C07281=1014.673,-56.612,386.212,-24.068,21.603,-43.637
C07282=1014.673,-56.279,386.186,-24.068,21.603,-43.632
C07283=1014.675,-55.946,386.161,-24.069,21.603,-43.627
C07284=1014.675,-55.613,386.136,-24.070,21.602,-43.623
C07285=1014.676,-55.280,386.111,-24.070,21.602,-43.618
C07286=1014.676,-54.948,386.085,-24.071,21.601,-43.613
C07287=1014.677,-54.616,386.060,-24.072,21.601,-43.608
C07288=1014.678,-54.284,386.034,-24.072,21.600,-43.603
C07289=1014.679,-53.951,386.010,-24.073,21.599,-43.599
C07290=1014.679,-53.619,385.984,-24.074,21.600,-43.594
C07291=1014.680,-53.287,385.959,-24.074,21.598,-43.589
C07292=1014.680,-52.954,385.933,-24.075,21.598,-43.584
C07293=1014.681,-52.622,385.909,-24.075,21.597,-43.579
C07294=1014.681,-52.290,385.883,-24.076,21.597,-43.575
C07295=1014.682,-51.957,385.857,-24.077,21.597,-43.570
C07296=1014.683,-51.625,385.832,-24.077,21.596,-43.566
C07297=1014.683,-51.293,385.806,-24.078,21.596,-43.560
C07298=1014.683,-50.960,385.781,-24.079,21.595,-43.555
C07299=1014.684,-50.628,385.756,-24.079,21.594,-43.551
C07300=1014.684,-50.296,385.731,-24.080,21.595,-43.546
C07301=1014.685,-49.963,385.705,-24.080,21.593,-43.542
C07302=1014.685,-49.630,385.680,-24.081,21.593,-43.536
C07303=1014.686,-49.298,385.654,-24.081,21.592,-43.532
C07304=1014.686,-48.966,385.629,-24.082,21.592,-43.527
C07305=1014.686,-48.633,385.604,-24.083,21.592,-43.522
C07306=1014.686,-48.301,385.578,-24.083,21.591,-43.518
C07307=1014.687,-47.968,385.552,-24.084,21.591,-43.512
C07308=1014.687,-47.635,385.527,-24.085,21.589,-43.508
C07309=1014.687,-47.303,385.501,-24.086,21.589,-43.503
C07310=1014.688,-46.971,385.476,-24.086,21.590,-43.498
C07311=1014.688,-46.639,385.450,-24.087,21.588,-43.494
C07312=1014.688,-46.306,385.425,-24.088,21.588,-43.488
C07313=1014.689,-45.973,385.399,-24.088,21.588,-43.485
C07314=1014.689,-45.641,385.373,-24.089,21.587,-43.479
C07315=1014.689,-45.308,385.348,-24.089,21.586,-43.475
C07316=1014.689,-44.976,385.323,-24.090,21.586,-43.470
C07317=1014.688,-44.643,385.296,-24.091,21.586,-43.465
C07318=1014.688,-44.310,385.271,-24.091,21.585,-43.461
C07319=1014.689,-43.978,385.246,-24.092,21.585,-43.455
C07320=1014.689,-43.645,385.220,-24.092,21.584,-43.451
C07321=1014.689,-43.312,385.195,-24.093,21.583,-43.446
C07322=1014.689,-42.980,385.168,-24.094,21.583,-43.442
C07323=1014.689,-42.648,385.143,-24.094,21.583,-43.437
C07324=1014.689,-42.315,385.118,-24.095,21.582,-43.431
C07325=1014.688,-41.982,385.091,-24.096,21.582,-43.427
C07326=1014.689,-41.650,385.066,-24.096,21.582,-43.422
C07327=1014.689,-41.317,385.041,-24.097,21.580,-43.418
C07328=1014.688,-40.985,385.015,-24.098,21.580,-43.413
C07329=1014.689,-40.652,384.988,-24.098,21.580,-43.409
C07330=1014.688,-40.319,384.963,-24.099,21.579,-43.404
C07331=1014.688,-39.987,384.937,-24.100,21.579,-43.398
C07332=1014.688,-39.654,384.911,-24.100,21.578,-43.394
C07333=1014.688,-39.321,384.886,-24.101,21.578,-43.389
C07334=1014.687,-38.989,384.860,-24.101,21.577,-43.385
C07335=1014.687,-38.657,384.834,-24.102,21.577,-43.380
C07336=1014.687,-38.323,384.808,-24.102,21.576,-43.376
C07337=1014.687,-37.991,384.783,-24.103,21.576,-43.371
C07338=1014.686,-37.658,384.757,-24.104,21.575,-43.366
C07339=1014.686,-37.326,384.731,-24.105,21.575,-43.361
C07340=1014.686,-36.993,384.705,-24.105,21.574,-43.357
C07341=1014.685,-36.660,384.680,-24.106,21.574,-43.352
C07342=1014.684,-36.328,384.653,-24.107,21.574,-43.347
C07343=1014.685,-35.995,384.628,-24.107,21.573,-43.343
C07344=1014.684,-35.662,384.602,-24.108,21.573,-43.337
C07345=1014.683,-35.330,384.576,-24.108,21.572,-43.334
C07346=1014.683,-34.997,384.549,-24.109,21.572,-43.328
C07347=1014.683,-34.664,384.525,-24.109,21.571,-43.324
C07348=1014.682,-34.332,384.498,-24.110,21.571,-43.319
C07349=1014.682,-33.999,384.472,-24.111,21.570,-43.315
C07350=1014.681,-33.666,384.446,-24.111,21.570,-43.310
C07351=1014.680,-33.334,384.420,-24.112,21.569,-43.306
C07352=1014.680,-33.001,384.395,-24.113,21.569,-43.301
C07353=1014.679,-32.668,384.368,-24.113,21.568,-43.296
C07354=1014.679,-32.336,384.342,-24.114,21.568,-43.291
C07355=1014.678,-32.002,384.316,-24.114,21.567,-43.287
C07356=1014.677,-31.670,384.290,-24.115,21.567,-43.282
C07357=1014.677,-31.337,384.264,-24.116,21.566,-43.278
C07358=1014.676,-31.004,384.238,-24.116,21.566,-43.273
C07359=1014.675,-30.672,384.212,-24.117,21.565,-43.269
C07360=1014.675,-30.339,384.186,-24.118,21.565,-43.264
C07361=1014.674,-30.006,384.160,-24.118,21.565,-43.260
C07362=1014.674,-29.674,384.134,-24.119,21.564,-43.254
C07363=1014.673,-29.340,384.108,-24.119,21.563,-43.250
C07364=1014.672,-29.008,384.081,-24.120,21.563,-43.245
C07365=1014.671,-28.675,384.055,-24.120,21.562,-43.241
C07366=1014.670,-28.342,384.030,-24.121,21.562,-43.236
C07367=1014.669,-28.010,384.004,-24.122,21.562,-43.232
C07368=1014.669,-27.678,383.977,-24.123,21.562,-43.227
C07369=1014.667,-27.344,383.951,-24.123,21.560,-43.223
C07370=1014.667,-27.012,383.925,-24.124,21.560,-43.217
C07371=1014.666,-26.679,383.899,-24.124,21.560,-43.214
C07372=1014.664,-26.346,383.872,-24.125,21.559,-43.208
C07373=1014.664,-26.013,383.846,-24.126,21.559,-43.204
C07374=1014.663,-25.680,383.821,-24.126,21.559,-43.199
C07375=1014.661,-25.348,383.794,-24.127,21.558,-43.195
C07376=1014.661,-25.015,383.768,-24.128,21.558,-43.190
C07377=1014.659,-24.682,383.742,-24.128,21.557,-43.186
C07378=1014.659,-24.349,383.715,-24.129,21.557,-43.181
C07379=1014.657,-24.017,383.688,-24.129,21.556,-43.177
C07380=1014.657,-23.683,383.663,-24.130,21.556,-43.171
C07381=1014.655,-23.351,383.636,-24.131,21.555,-43.168
C07382=1014.654,-23.018,383.611,-24.131,21.556,-43.162
C07383=1014.653,-22.685,383.584,-24.132,21.554,-43.158
C07384=1014.652,-22.353,383.558,-24.133,21.554,-43.153
C07385=1014.651,-22.019,383.531,-24.133,21.554,-43.149
C07386=1014.649,-21.687,383.505,-24.134,21.553,-43.144
C07387=1014.648,-21.355,383.479,-24.134,21.552,-43.140
C07388=1014.647,-21.021,383.453,-24.135,21.553,-43.135
C07389=1014.645,-20.689,383.426,-24.136,21.552,-43.131
C07390=1014.644,-20.356,383.400,-24.136,21.551,-43.127
C07391=1014.643,-20.023,383.374,-24.137,21.551,-43.122
C07392=1014.642,-19.851,383.360,-24.137,21.550,-43.118
C07393=1014.640,-19.434,383.327,-24.138,21.550,-43.112
C07394=1014.640,-19.187,383.307,-24.139,21.550,-43.109
C07395=1014.638,-18.925,383.286,-24.139,21.550,-43.107
C07396=1014.637,-18.663,383.266,-24.139,21.549,-43.105
C07397=1014.637,-18.416,383.246,-24.139,21.548,-43.103
C07398=1014.635,-18.194,383.228,-24.140,21.549,-43.100
C07399=1014.634,-17.829,383.200,-24.141,21.548,-43.092
C07400=1014.632,-17.496,383.173,-24.141,21.547,-43.088
C07401=1014.631,-17.163,383.146,-24.142,21.547,-43.083
C07402=1014.630,-16.830,383.120,-24.142,21.547,-43.079
C07403=1014.628,-16.497,383.093,-24.143,21.546,-43.074
C07404=1014.626,-16.162,383.067,-24.144,21.546,-43.070
C07405=1014.624,-15.827,383.040,-24.145,21.546,-43.065
C07406=1014.623,-15.491,383.014,-24.145,21.545,-43.061
C07407=1014.621,-15.152,382.986,-24.146,21.544,-43.055
C07408=1014.619,-14.812,382.960,-24.146,21.544,-43.052
C07409=1014.618,-14.471,382.932,-24.147,21.544,-43.046
C07410=1014.616,-14.127,382.905,-24.147,21.543,-43.042
C07411=1014.615,-13.780,382.877,-24.148,21.543,-43.037
C07412=1014.613,-13.432,382.849,-24.149,21.542,-43.033
C07413=1014.611,-13.081,382.822,-24.149,21.542,-43.028
C07414=1014.609,-12.729,382.793,-24.150,21.541,-43.024
C07415=1014.607,-12.376,382.765,-24.151,21.541,-43.019
C07416=1014.606,-12.021,382.737,-24.151,21.540,-43.014
C07417=1014.604,-11.664,382.708,-24.152,21.540,-43.009
C07418=1014.602,-11.306,382.680,-24.152,21.539,-43.006
C07419=1014.599,-10.948,382.651,-24.153,21.539,-43.000
C07420=1014.598,-10.588,382.623,-24.154,21.539,-42.995
C07421=1014.596,-10.227,382.593,-24.154,21.538,-42.991
C07422=1014.594,-9.866,382.564,-24.155,21.538,-42.985
C07423=1014.592,-9.504,382.535,-24.156,21.537,-42.982
C07424=1014.589,-9.142,382.506,-24.156,21.536,-42.976
C07425=1014.587,-8.778,382.477,-24.157,21.536,-42.971
C07426=1014.585,-8.416,382.448,-24.158,21.536,-42.967
C07427=1014.583,-8.053,382.419,-24.158,21.535,-42.961
C07428=1014.580,-7.686,382.390,-24.159,21.535,-42.956
C07429=1014.578,-7.317,382.361,-24.160,21.534,-42.952
C07430=1014.576,-6.945,382.330,-24.160,21.534,-42.947
C07431=1014.574,-6.571,382.300,-24.161,21.533,-42.941
C07432=1014.572,-6.196,382.270,-24.162,21.533,-42.937
C07433=1014.568,-5.820,382.240,-24.163,21.533,-42.932
C07434=1014.567,-5.447,382.210,-24.163,21.532,-42.928
C07435=1014.564,-5.076,382.180,-24.164,21.532,-42.923
C07436=1014.561,-4.710,382.150,-24.164,21.531,-42.919
C07437=1014.559,-4.349,382.122,-24.165,21.530,-42.913
C07438=1014.556,-3.991,382.092,-24.166,21.531,-42.908
C07439=1014.554,-3.637,382.065,-24.166,21.529,-42.904
C07440=1014.552,-3.285,382.036,-24.167,21.529,-42.899
C07441=1014.549,-2.933,382.007,-24.167,21.529,-42.895
C07442=1014.547,-2.583,381.979,-24.168,21.529,-42.890
C07443=1014.545,-2.236,381.951,-24.169,21.528,-42.886
C07444=1014.542,-1.888,381.923,-24.169,21.528,-42.880
C07445=1014.540,-1.544,381.896,-24.170,21.527,-42.877
C07446=1014.537,-1.201,381.868,-24.170,21.527,-42.873
C07447=1014.535,-0.858,381.840,-24.171,21.526,-42.867
C07448=1014.532,-0.519,381.813,-24.172,21.526,-42.864
C07449=1014.529,-0.180,381.785,-24.172,21.526,-42.858
C07450=1014.527,0.157,381.759,-24.173,21.525,-42.855
C07451=1014.525,0.493,381.731,-24.173,21.525,-42.851
C07452=1014.522,0.827,381.704,-24.174,21.525,-42.846
C07453=1014.519,1.161,381.677,-24.175,21.524,-42.842
C07454=1014.516,1.495,381.650,-24.175,21.523,-42.838
C07455=1014.514,1.825,381.623,-24.176,21.523,-42.834
C07456=1014.512,2.138,381.598,-24.176,21.523,-42.831
C07457=1014.509,2.426,381.574,-24.177,21.522,-42.827
C07458=1014.508,2.695,381.553,-24.177,21.522,-42.823
C07459=1014.505,2.957,381.532,-24.178,21.522,-42.818
C07460=1014.503,3.226,381.510,-24.179,21.521,-42.814
C07461=1014.500,3.515,381.487,-24.179,21.521,-42.810
C07462=1014.498,3.829,381.461,-24.179,21.520,-42.807
C07463=1014.496,4.158,381.434,-24.180,21.521,-42.803
C07464=1014.493,4.490,381.408,-24.180,21.519,-42.799
C07465=1014.490,4.821,381.380,-24.181,21.519,-42.795
C07466=1014.487,5.151,381.354,-24.181,21.518,-42.792
C07467=1014.485,5.481,381.327,-24.182,21.519,-42.786
C07468=1014.481,5.811,381.300,-24.183,21.518,-42.783
C07469=1014.479,6.141,381.273,-24.183,21.518,-42.779
C07470=1014.475,6.470,381.247,-24.184,21.518,-42.774
C07471=1014.473,6.798,381.220,-24.185,21.517,-42.770
C07472=1014.470,7.126,381.193,-24.185,21.517,-42.766
C07473=1014.467,7.451,381.167,-24.186,21.516,-42.762
C07474=1014.464,7.775,381.141,-24.186,21.516,-42.759
C07475=1014.462,8.095,381.114,-24.186,21.515,-42.755
C07476=1014.459,8.413,381.088,-24.187,21.516,-42.750
C07477=1014.456,8.729,381.063,-24.188,21.515,-42.746
C07478=1014.453,9.044,381.037,-24.188,21.515,-42.742
C07479=1014.450,9.359,381.011,-24.189,21.514,-42.738
C07480=1014.448,9.673,380.986,-24.190,21.514,-42.733
C07481=1014.444,9.989,380.961,-24.190,21.514,-42.730
C07482=1014.442,10.306,380.934,-24.191,21.513,-42.726
C07483=1014.438,10.625,380.909,-24.191,21.513,-42.722
C07484=1014.435,10.945,380.883,-24.192,21.512,-42.718
C07485=1014.432,11.267,380.856,-24.192,21.512,-42.715
C07486=1014.429,11.591,380.830,-24.193,21.511,-42.711
C07487=1014.426,11.914,380.803,-24.193,21.511,-42.707
C07488=1014.423,12.237,380.777,-24.194,21.511,-42.702
C07489=1014.420,12.561,380.751,-24.194,21.510,-42.698
C07490=1014.416,12.885,380.724,-24.195,21.510,-42.694
C07491=1014.413,13.208,380.698,-24.195,21.509,-42.691
C07492=1014.410,13.533,380.671,-24.196,21.509,-42.687
C07493=1014.406,13.857,380.645,-24.197,21.509,-42.682
C07494=1014.403,14.181,380.618,-24.197,21.509,-42.678
C07495=1014.400,14.506,380.591,-24.198,21.508,-42.674
C07496=1014.396,14.832,380.566,-24.198,21.508,-42.670
C07497=1014.393,15.158,380.539,-24.199,21.507,-42.667
C07498=1014.390,15.484,380.512,-24.199,21.507,-42.663
C07499=1014.387,15.811,380.485,-24.200,21.507,-42.658
C07500=1014.383,16.139,380.458,-24.200,21.506,-42.654
C07501=1014.380,16.467,380.431,-24.201,21.506,-42.650
C07502=1014.376,16.795,380.405,-24.201,21.505,-42.646
C07503=1014.372,17.124,380.378,-24.202,21.505,-42.643
C07504=1014.370,17.454,380.351,-24.202,21.504,-42.639
C07505=1014.366,17.784,380.324,-24.203,21.504,-42.634
C07506=1014.362,18.115,380.296,-24.204,21.504,-42.630
C07507=1014.358,18.446,380.270,-24.204,21.503,-42.626
C07508=1014.354,18.778,380.243,-24.205,21.503,-42.622
C07509=1014.352,19.110,380.215,-24.205,21.502,-42.619
C07510=1014.347,19.458,380.187,-24.206,21.503,-42.613
C07511=1014.342,19.875,380.152,-24.207,21.502,-42.608
C07512=1014.340,20.112,380.133,-24.207,21.502,-42.604
C07513=1014.338,20.358,380.113,-24.207,21.502,-42.603
C07514=1014.334,20.606,380.093,-24.208,21.502,-42.601
C07515=1014.332,20.848,380.073,-24.208,21.502,-42.599
C07516=1014.329,21.075,380.054,-24.208,21.501,-42.597
C07517=1014.327,21.282,380.037,-24.209,21.501,-42.593
C07518=1014.322,21.639,380.008,-24.209,21.500,-42.588
C07519=1014.319,21.962,379.981,-24.210,21.501,-42.584
C07520=1014.315,22.256,379.957,-24.210,21.500,-42.582
C07521=1014.312,22.509,379.936,-24.210,21.499,-42.580
C07522=1014.307,22.919,379.903,-24.211,21.499,-42.573
C07523=1014.303,23.327,379.869,-24.212,21.498,-42.565
C07524=1014.300,23.579,379.849,-24.213,21.498,-42.562
C07525=1014.296,23.873,379.825,-24.213,21.498,-42.560
C07526=1014.292,24.200,379.798,-24.213,21.497,-42.558
C07527=1014.288,24.534,379.770,-24.214,21.497,-42.553
C07528=1014.284,24.868,379.742,-24.215,21.497,-42.549
C07529=1014.280,25.202,379.715,-24.215,21.496,-42.545
C07530=1014.276,25.537,379.688,-24.216,21.496,-42.541
C07531=1014.271,25.870,379.660,-24.216,21.495,-42.538
C07532=1014.268,26.205,379.632,-24.217,21.495,-42.534
C07533=1014.263,26.539,379.605,-24.217,21.494,-42.530
C07534=1014.259,26.873,379.577,-24.218,21.494,-42.525
C07535=1014.254,27.208,379.550,-24.219,21.495,-42.522
C07536=1014.251,27.542,379.522,-24.219,21.494,-42.518
C07537=1014.246,27.876,379.495,-24.220,21.494,-42.514
C07538=1014.242,28.211,379.468,-24.220,21.493,-42.510
C07539=1014.238,28.545,379.440,-24.221,21.493,-42.507
C07540=1014.233,28.879,379.413,-24.221,21.492,-42.503
C07541=1014.229,29.214,379.385,-24.222,21.493,-42.498
C07542=1014.224,29.548,379.358,-24.222,21.492,-42.494
C07543=1014.220,29.882,379.330,-24.223,21.492,-42.490
C07544=1014.216,30.216,379.302,-24.223,21.491,-42.486
C07545=1014.211,30.551,379.274,-24.224,21.491,-42.483
C07546=1014.207,30.885,379.247,-24.224,21.490,-42.479
C07547=1014.203,31.220,379.220,-24.225,21.490,-42.475
C07548=1014.197,31.555,379.192,-24.225,21.489,-42.471
C07549=1014.193,31.888,379.165,-24.226,21.489,-42.468
C07550=1014.189,32.224,379.137,-24.226,21.489,-42.464
C07551=1014.184,32.558,379.109,-24.227,21.489,-42.459
C07552=1014.180,32.893,379.082,-24.228,21.489,-42.455
C07553=1014.174,33.227,379.054,-24.228,21.488,-42.452
C07554=1014.170,33.561,379.027,-24.229,21.488,-42.448
C07555=1014.165,33.896,378.999,-24.229,21.487,-42.444
C07556=1014.161,34.230,378.971,-24.230,21.487,-42.440
C07557=1014.155,34.565,378.944,-24.230,21.486,-42.437
C07558=1014.151,34.899,378.915,-24.231,21.486,-42.433
C07559=1014.146,35.234,378.889,-24.231,21.485,-42.429
C07560=1014.141,35.569,378.861,-24.232,21.486,-42.426
C07561=1014.136,35.903,378.834,-24.232,21.485,-42.422
C07562=1014.131,36.237,378.806,-24.233,21.485,-42.418
C07563=1014.126,36.573,378.778,-24.234,21.485,-42.413
C07564=1014.121,36.907,378.750,-24.234,21.485,-42.409
C07565=1014.117,37.241,378.723,-24.235,21.484,-42.405
C07566=1014.112,37.576,378.695,-24.235,21.484,-42.402
C07567=1014.106,37.911,378.668,-24.236,21.483,-42.398
C07568=1014.101,38.246,378.640,-24.236,21.483,-42.395
C07569=1014.096,38.580,378.612,-24.237,21.483,-42.391
C07570=1014.092,38.915,378.585,-24.237,21.483,-42.387
C07571=1014.086,39.249,378.557,-24.238,21.482,-42.383
C07572=1014.081,39.584,378.530,-24.238,21.482,-42.380
C07573=1014.076,39.919,378.502,-24.239,21.481,-42.376
C07574=1014.071,40.253,378.474,-24.239,21.481,-42.372
C07575=1014.066,40.588,378.446,-24.240,21.481,-42.369
C07576=1014.060,40.923,378.419,-24.240,21.481,-42.365
C07577=1014.055,41.257,378.391,-24.241,21.480,-42.361
C07578=1014.049,41.592,378.364,-24.241,21.480,-42.357
C07579=1014.045,41.927,378.336,-24.242,21.479,-42.354
C07580=1014.038,42.262,378.308,-24.242,21.479,-42.350
C07581=1014.033,42.596,378.280,-24.243,21.479,-42.347
C07582=1014.028,42.931,378.252,-24.243,21.479,-42.343
C07583=1014.022,43.265,378.225,-24.244,21.478,-42.339
C07584=1014.017,43.600,378.198,-24.244,21.478,-42.335
C07585=1014.012,43.935,378.170,-24.245,21.477,-42.332
C07586=1014.006,44.270,378.142,-24.245,21.477,-42.328
C07587=1014.001,44.605,378.114,-24.246,21.477,-42.325
C07588=1013.995,44.940,378.087,-24.246,21.477,-42.321
C07589=1013.989,45.275,378.059,-24.247,21.476,-42.317
C07590=1013.984,45.609,378.031,-24.247,21.476,-42.313
C07591=1013.978,45.944,378.004,-24.248,21.475,-42.309
C07592=1013.972,46.279,377.976,-24.248,21.475,-42.306
C07593=1013.967,46.613,377.948,-24.249,21.475,-42.302
C07594=1013.961,46.948,377.921,-24.249,21.475,-42.299
C07595=1013.955,47.283,377.893,-24.250,21.474,-42.295
C07596=1013.950,47.618,377.865,-24.250,21.474,-42.291
C07597=1013.943,47.953,377.837,-24.251,21.473,-42.287
C07598=1013.938,48.287,377.810,-24.251,21.473,-42.284
C07599=1013.932,48.623,377.782,-24.252,21.473,-42.280
C07600=1013.926,48.957,377.755,-24.252,21.473,-42.277
C07601=1013.920,49.292,377.727,-24.253,21.472,-42.273
C07602=1013.913,49.627,377.699,-24.253,21.472,-42.269
C07603=1013.908,49.961,377.672,-24.254,21.472,-42.266
C07604=1013.902,50.296,377.644,-24.254,21.471,-42.262
C07605=1013.896,50.631,377.616,-24.255,21.471,-42.258
C07606=1013.890,50.966,377.589,-24.255,21.471,-42.254
C07607=1013.884,51.301,377.561,-24.256,21.471,-42.251
C07608=1013.877,51.636,377.533,-24.256,21.470,-42.247
C07609=1013.871,51.970,377.506,-24.257,21.470,-42.244
C07610=1013.865,52.305,377.478,-24.257,21.470,-42.240
C07611=1013.859,52.641,377.450,-24.258,21.469,-42.238
C07612=1013.852,52.975,377.423,-24.258,21.469,-42.234
C07613=1013.846,53.310,377.395,-24.259,21.468,-42.230
C07614=1013.840,53.645,377.367,-24.259,21.468,-42.227
C07615=1013.816,54.896,377.264,-24.271,21.503,-42.191
C07616=1013.815,54.977,377.257,-24.281,21.541,-42.167
C07617=1013.807,55.373,377.225,-24.331,21.722,-42.052
C07618=1013.799,55.768,377.192,-24.380,21.904,-41.938
C07619=1013.792,56.164,377.159,-24.428,22.086,-41.824
C07620=1013.784,56.560,377.127,-24.477,22.269,-41.710
C07621=1013.776,56.955,377.094,-24.525,22.453,-41.598
C07622=1013.769,57.351,377.061,-24.572,22.637,-41.485
C07623=1013.760,57.747,377.029,-24.620,22.823,-41.372
C07624=1013.753,58.143,376.996,-24.667,23.008,-41.261
C07625=1013.745,58.538,376.963,-24.715,23.195,-41.149
C07626=1013.737,58.934,376.931,-24.761,23.381,-41.038
C07627=1013.730,59.330,376.898,-24.808,23.569,-40.927
C07628=1013.722,59.726,376.866,-24.853,23.757,-40.818
C07629=1013.714,60.121,376.833,-24.899,23.946,-40.708
C07630=1013.706,60.518,376.801,-24.945,24.135,-40.598
C07631=1013.699,60.913,376.768,-24.990,24.326,-40.489
C07632=1013.690,61.309,376.736,-25.035,24.517,-40.381
C07633=1013.683,61.704,376.704,-25.080,24.707,-40.272
C07634=1013.675,62.102,376.671,-25.124,24.901,-40.164
C07635=1013.669,62.386,376.647,-25.156,25.038,-40.089
C07636=1013.665,62.605,376.629,-25.180,25.145,-40.028
C07637=1013.659,62.847,376.610,-25.207,25.264,-39.964
C07638=1013.654,63.095,376.589,-25.234,25.384,-39.898
C07639=1013.650,63.330,376.570,-25.260,25.499,-39.835
C07640=1013.646,63.542,376.553,-25.283,25.603,-39.779
C07641=1013.643,63.947,376.517,-25.297,25.665,-39.741
C07642=1013.642,64.165,376.495,-25.299,25.671,-39.736
C07643=1013.641,64.392,376.475,-25.300,25.677,-39.731
C07644=1013.641,64.619,376.454,-25.302,25.682,-39.725
C07645=1013.640,64.840,376.432,-25.303,25.688,-39.721
C07646=1013.639,65.060,376.413,-25.304,25.693,-39.715
C07647=1013.638,65.275,376.392,-25.306,25.699,-39.711
C07648=1013.638,65.483,376.373,-25.307,25.703,-39.706
C07649=1013.637,65.875,376.335,-25.310,25.713,-39.697
C07650=1013.635,66.203,376.304,-25.312,25.721,-39.689
C07651=1013.634,66.566,376.270,-25.314,25.731,-39.681
C07652=1013.633,66.963,376.233,-25.317,25.740,-39.672
C07653=1013.631,67.362,376.196,-25.319,25.750,-39.663
C07654=1013.630,67.763,376.158,-25.322,25.760,-39.654
C07655=1013.628,68.173,376.120,-25.325,25.771,-39.645
C07656=1013.626,68.591,376.080,-25.328,25.781,-39.635
C07657=1013.626,69.007,376.041,-25.330,25.792,-39.626
C07658=1013.624,69.416,376.002,-25.333,25.803,-39.615
C07659=1013.622,69.819,375.964,-25.336,25.813,-39.606
C07660=1013.621,70.224,375.926,-25.338,25.823,-39.597
C07661=1013.620,70.628,375.888,-25.341,25.832,-39.588
C07662=1013.618,71.032,375.849,-25.343,25.843,-39.579
C07663=1013.617,71.437,375.812,-25.346,25.854,-39.569
C07664=1013.616,71.842,375.773,-25.349,25.865,-39.560
C07665=1013.614,72.248,375.735,-25.352,25.876,-39.550
C07666=1013.612,72.656,375.696,-25.354,25.886,-39.541
C07667=1013.611,73.065,375.657,-25.357,25.896,-39.532
C07668=1013.609,73.476,375.618,-25.360,25.907,-39.522
C07669=1013.608,73.891,375.579,-25.363,25.919,-39.512
C07670=1013.608,74.110,375.558,-25.364,25.923,-39.507
C07671=1013.606,74.338,375.536,-25.366,25.931,-39.502
C07672=1013.606,74.565,375.514,-25.367,25.936,-39.498
C07673=1013.605,74.780,375.495,-25.369,25.941,-39.492
C07674=1013.605,74.989,375.475,-25.370,25.947,-39.488
C07675=1013.603,75.403,375.435,-25.373,25.958,-39.477
C07676=1013.601,75.812,375.397,-25.376,25.970,-39.467
C07677=1013.600,76.214,375.358,-25.378,25.980,-39.458
C07678=1013.599,76.607,375.321,-25.381,25.990,-39.450
C07679=1013.597,76.994,375.284,-25.384,26.001,-39.441
C07680=1013.595,77.376,375.247,-25.386,26.011,-39.432
C07681=1013.594,77.757,375.211,-25.389,26.022,-39.423
C07682=1013.593,78.141,375.175,-25.392,26.033,-39.413
C07683=1013.591,78.530,375.138,-25.394,26.043,-39.404
C07684=1013.590,78.925,375.100,-25.397,26.053,-39.395
C07685=1013.588,79.326,375.061,-25.400,26.065,-39.385
C07686=1013.586,79.735,375.023,-25.402,26.076,-39.377
C07687=1013.585,80.147,374.983,-25.405,26.087,-39.367
C07688=1013.584,80.530,374.947,-25.408,26.098,-39.358
C07689=1013.582,80.893,374.912,-25.410,26.108,-39.349
C07690=1013.580,81.287,374.874,-25.413,26.119,-39.340
C07691=1013.579,81.701,374.835,-25.416,26.131,-39.330
C07692=1013.577,82.115,374.795,-25.419,26.143,-39.321
C07693=1013.576,82.528,374.755,-25.422,26.154,-39.311
C07694=1013.574,82.940,374.717,-25.425,26.165,-39.300
C07695=1013.572,83.351,374.677,-25.428,26.177,-39.291
C07696=1013.571,83.760,374.637,-25.431,26.189,-39.281
C07697=1013.569,84.168,374.599,-25.433,26.200,-39.272
C07698=1013.567,84.575,374.559,-25.436,26.212,-39.263
C07699=1013.566,84.981,374.521,-25.439,26.224,-39.253
C07700=1013.565,85.385,374.482,-25.442,26.236,-39.243
C07701=1013.563,85.788,374.442,-25.445,26.248,-39.233
C07702=1013.561,86.189,374.404,-25.447,26.259,-39.225
C07703=1013.560,86.591,374.366,-25.450,26.271,-39.215
C07704=1013.559,86.989,374.327,-25.453,26.283,-39.205
C07705=1013.557,87.383,374.290,-25.456,26.294,-39.197
C07706=1013.555,87.768,374.252,-25.459,26.305,-39.186
C07707=1013.554,88.145,374.215,-25.461,26.316,-39.178
C07708=1013.552,88.520,374.179,-25.464,26.328,-39.168
C07709=1013.551,88.898,374.143,-25.467,26.338,-39.159
C07710=1013.549,89.283,374.106,-25.469,26.349,-39.151
C07711=1013.548,89.679,374.067,-25.472,26.361,-39.141
C07712=1013.546,89.913,374.044,-25.474,26.367,-39.135
C07713=1013.546,90.188,374.018,-25.475,26.375,-39.130
C07714=1013.544,90.468,373.991,-25.477,26.382,-39.124
C07715=1013.543,90.713,373.967,-25.479,26.390,-39.119
C07716=1013.542,91.115,373.928,-25.482,26.402,-39.109
C07717=1013.540,91.510,373.890,-25.485,26.413,-39.099
C07718=1013.538,91.905,373.852,-25.488,26.427,-39.088
C07719=1013.537,92.300,373.814,-25.491,26.440,-39.079
C07720=1013.535,92.694,373.775,-25.494,26.452,-39.069
C07721=1013.533,93.088,373.737,-25.497,26.464,-39.060
C07722=1013.531,93.483,373.699,-25.499,26.475,-39.051
C07723=1013.530,93.877,373.661,-25.502,26.485,-39.042
C07724=1013.528,94.272,373.622,-25.504,26.496,-39.034
C07725=1013.528,94.666,373.584,-25.507,26.508,-39.024
C07726=1013.526,95.061,373.545,-25.510,26.521,-39.014
C07727=1013.524,95.455,373.508,-25.513,26.533,-39.005
C07728=1013.522,95.849,373.469,-25.516,26.547,-38.994
C07729=1013.520,96.244,373.430,-25.520,26.561,-38.984
C07730=1013.519,96.638,373.392,-25.522,26.573,-38.974
C07731=1013.517,97.033,373.354,-25.525,26.584,-38.965
C07732=1013.516,97.427,373.316,-25.528,26.595,-38.957
C07733=1013.514,97.822,373.277,-25.530,26.607,-38.947
C07734=1013.512,98.216,373.238,-25.533,26.619,-38.938
C07735=1013.511,98.611,373.200,-25.536,26.631,-38.928
C07736=1013.508,99.004,373.162,-25.539,26.646,-38.918
C07737=1013.507,99.398,373.123,-25.543,26.659,-38.907
C07738=1013.505,99.793,373.085,-25.546,26.673,-38.898
C07739=1013.504,100.188,373.046,-25.548,26.683,-38.889
C07740=1013.502,100.581,373.008,-25.551,26.695,-38.880
C07741=1013.500,100.976,372.969,-25.554,26.707,-38.872
C07742=1013.499,101.370,372.930,-25.556,26.719,-38.862
C07743=1013.497,101.765,372.891,-25.560,26.733,-38.851
C07744=1013.495,102.159,372.854,-25.562,26.746,-38.842
C07745=1013.493,102.553,372.814,-25.566,26.760,-38.832
C07746=1013.492,102.947,372.775,-25.569,26.774,-38.822
C07747=1013.490,103.342,372.738,-25.572,26.786,-38.812
C07748=1013.488,103.736,372.699,-25.574,26.798,-38.803
C07749=1013.486,104.130,372.660,-25.577,26.810,-38.794
C07750=1013.485,104.524,372.621,-25.580,26.822,-38.784
C07751=1013.483,104.919,372.582,-25.583,26.835,-38.775
C07752=1013.482,105.312,372.544,-25.586,26.850,-38.765
C07753=1013.480,105.707,372.505,-25.589,26.864,-38.755
C07754=1013.478,106.101,372.466,-25.593,26.878,-38.744
C07755=1013.476,106.496,372.427,-25.595,26.891,-38.735
C07756=1013.474,106.889,372.388,-25.598,26.903,-38.725
C07757=1013.473,107.283,372.350,-25.601,26.914,-38.717
C07758=1013.471,107.678,372.311,-25.604,26.927,-38.708
C07759=1013.470,108.072,372.272,-25.607,26.941,-38.697
C07760=1013.467,108.466,372.233,-25.610,26.954,-38.688
C07761=1013.466,108.860,372.194,-25.613,26.969,-38.678
C07762=1013.464,109.254,372.155,-25.616,26.984,-38.666
C07763=1013.462,109.648,372.116,-25.619,26.998,-38.658
C07764=1013.461,110.042,372.078,-25.622,27.010,-38.648
C07765=1013.459,110.436,372.038,-25.625,27.023,-38.639
C07766=1013.457,110.831,371.999,-25.628,27.035,-38.629
C07767=1013.455,111.224,371.961,-25.631,27.048,-38.620
C07768=1013.454,111.619,371.922,-25.634,27.062,-38.609
C07769=1013.452,112.013,371.882,-25.637,27.076,-38.599
C07770=1013.450,112.407,371.843,-25.640,27.092,-38.589
C07771=1013.448,112.801,371.805,-25.644,27.106,-38.579
C07772=1013.446,113.195,371.766,-25.646,27.119,-38.570
C07773=1013.445,113.590,371.727,-25.649,27.132,-38.561
C07774=1013.443,113.984,371.687,-25.652,27.145,-38.551
C07775=1013.441,114.378,371.648,-25.655,27.157,-38.542
C07776=1013.439,114.772,371.610,-25.658,27.172,-38.532
C07777=1013.438,115.166,371.570,-25.661,27.186,-38.522
C07778=1013.436,115.560,371.531,-25.664,27.201,-38.512
C07779=1013.434,115.954,371.492,-25.668,27.217,-38.500
C07780=1013.432,116.348,371.453,-25.671,27.230,-38.491
C07781=1013.430,116.742,371.414,-25.674,27.243,-38.482
C07782=1013.429,117.136,371.374,-25.676,27.256,-38.473
C07783=1013.426,117.531,371.334,-25.680,27.270,-38.463
C07784=1013.425,117.925,371.295,-25.682,27.284,-38.454
C07785=1013.422,118.319,371.257,-25.686,27.298,-38.444
C07786=1013.421,118.713,371.218,-25.689,27.313,-38.432
C07787=1013.419,119.107,371.178,-25.692,27.329,-38.422
C07788=1013.418,119.501,371.139,-25.695,27.343,-38.412
C07789=1013.416,119.895,371.100,-25.698,27.356,-38.403
C07790=1013.414,120.289,371.059,-25.701,27.370,-38.394
C07791=1013.412,120.683,371.020,-25.704,27.383,-38.384
C07792=1013.410,121.077,370.981,-25.707,27.397,-38.375
C07793=1013.409,121.471,370.942,-25.710,27.412,-38.365
C07794=1013.407,121.865,370.902,-25.714,27.428,-38.354
C07795=1013.405,122.260,370.863,-25.717,27.443,-38.344
C07796=1013.403,122.654,370.824,-25.720,27.459,-38.333
C07797=1013.401,123.048,370.784,-25.723,27.472,-38.324
C07798=1013.399,123.442,370.745,-25.726,27.486,-38.315
C07799=1013.397,123.836,370.705,-25.729,27.500,-38.304
C07800=1013.395,124.230,370.666,-25.732,27.513,-38.295
C07801=1013.394,124.625,370.627,-25.735,27.529,-38.286
C07802=1013.392,125.019,370.586,-25.738,27.544,-38.274
C07803=1013.390,125.413,370.547,-25.742,27.560,-38.265
C07804=1013.388,125.807,370.508,-25.745,27.576,-38.254
C07805=1013.386,126.201,370.468,-25.748,27.591,-38.244
C07806=1013.384,126.596,370.429,-25.751,27.604,-38.235
C07807=1013.383,126.989,370.389,-25.754,27.618,-38.226
C07808=1013.381,127.384,370.349,-25.757,27.632,-38.216
C07809=1013.379,127.778,370.309,-25.760,27.647,-38.206
C07810=1013.377,128.172,370.270,-25.763,27.664,-38.195
C07811=1013.376,128.566,370.230,-25.767,27.679,-38.185
C07812=1013.374,128.960,370.191,-25.770,27.695,-38.174
C07813=1013.372,129.354,370.150,-25.773,27.711,-38.165
C07814=1013.370,129.749,370.111,-25.776,27.725,-38.155
C07815=1013.368,130.143,370.071,-25.779,27.738,-38.145
C07816=1013.366,130.537,370.032,-25.782,27.753,-38.136
C07817=1013.364,130.931,369.991,-25.785,27.768,-38.126
C07818=1013.362,131.326,369.952,-25.789,27.784,-38.115
C07819=1013.360,131.720,369.912,-25.792,27.800,-38.105
C07820=1013.359,132.114,369.873,-25.795,27.816,-38.094
C07821=1013.357,132.508,369.832,-25.799,27.834,-38.084
C07822=1013.355,132.902,369.793,-25.802,27.847,-38.075
C07823=1013.353,133.297,369.753,-25.805,27.862,-38.065
C07824=1013.351,133.692,369.713,-25.808,27.876,-38.055
C07825=1013.350,134.085,369.673,-25.811,27.892,-38.045
C07826=1013.347,134.480,369.633,-25.814,27.908,-38.034
C07827=1013.347,134.710,369.610,-25.816,27.917,-38.028
C07828=1013.345,134.970,369.583,-25.818,27.928,-38.022
C07829=1013.344,135.380,369.542,-25.822,27.946,-38.010
C07830=1013.342,135.749,369.505,-25.825,27.961,-38.000
C07831=1013.340,136.089,369.470,-25.828,27.975,-37.992
C07832=1013.338,136.410,369.438,-25.830,27.987,-37.984
C07833=1013.337,136.731,369.405,-25.833,28.001,-37.975
C07834=1013.336,137.074,369.370,-25.836,28.014,-37.966
C07835=1013.334,137.423,369.335,-25.839,28.029,-37.958
C07836=1013.332,137.723,369.304,-25.841,28.040,-37.950
C07837=1013.330,138.119,369.264,-25.844,28.056,-37.940
C07838=1013.330,138.338,369.242,-25.846,28.065,-37.934
C07839=1013.328,138.573,369.218,-25.848,28.074,-37.929
C07840=1013.327,138.822,369.192,-25.850,28.085,-37.922
C07841=1013.326,139.080,369.166,-25.852,28.095,-37.916
C07842=1013.324,139.342,369.140,-25.854,28.105,-37.909
C07843=1013.323,139.604,369.113,-25.856,28.116,-37.902
C07844=1013.322,139.857,369.088,-25.858,28.126,-37.896
C07845=1013.321,140.099,369.062,-25.861,28.137,-37.889
C07846=1013.320,140.325,369.039,-25.862,28.146,-37.883
C07847=1013.319,140.536,369.019,-25.864,28.154,-37.878
C07848=1013.318,140.754,368.996,-25.866,28.163,-37.872
C07849=1013.316,141.159,368.955,-25.869,28.180,-37.862
C07850=1013.315,141.424,368.928,-25.871,28.190,-37.855
C07851=1013.314,141.624,368.908,-25.873,28.198,-37.850
C07852=1013.312,142.025,368.866,-25.876,28.215,-37.839
C07853=1013.310,142.426,368.825,-25.880,28.232,-37.829
C07854=1013.308,142.829,368.784,-25.883,28.248,-37.820
C07855=1013.306,143.231,368.743,-25.886,28.264,-37.809
C07856=1013.304,143.634,368.702,-25.890,28.281,-37.798
C07857=1013.302,144.037,368.661,-25.893,28.298,-37.788
C07858=1013.300,144.442,368.620,-25.896,28.315,-37.777
C07859=1013.298,144.847,368.578,-25.900,28.332,-37.766
C07860=1013.297,145.252,368.536,-25.903,28.349,-37.756
C07861=1013.295,145.657,368.495,-25.906,28.366,-37.745
C07862=1013.293,146.063,368.454,-25.910,28.383,-37.735
C07863=1013.291,146.468,368.412,-25.913,28.400,-37.725
C07864=1013.290,146.877,368.371,-25.916,28.417,-37.714
C07865=1013.778,146.956,368.043,-24.372,21.404,-41.418
C07866=1013.780,146.610,368.078,-24.372,21.404,-41.420
C07867=1013.783,146.263,368.113,-24.372,21.404,-41.424
C07868=1013.783,145.917,368.149,-24.371,21.405,-41.425
C07869=1013.785,145.571,368.184,-24.371,21.405,-41.427
C07870=1013.787,145.226,368.220,-24.371,21.404,-41.431
C07871=1013.789,144.880,368.255,-24.370,21.405,-41.432
C07872=1013.790,144.536,368.291,-24.370,21.406,-41.435
C07873=1013.792,144.190,368.326,-24.370,21.405,-41.438
C07874=1013.793,143.846,368.362,-24.369,21.405,-41.440
C07875=1013.795,143.503,368.396,-24.369,21.406,-41.442
C07876=1013.797,143.160,368.431,-24.369,21.405,-41.445
C07877=1013.798,142.817,368.467,-24.368,21.406,-41.448
C07878=1013.800,142.475,368.502,-24.368,21.407,-41.449
C07879=1013.801,142.134,368.536,-24.368,21.406,-41.453
C07880=1013.803,141.794,368.571,-24.367,21.406,-41.455
C07881=1013.804,141.453,368.606,-24.367,21.407,-41.457
C07882=1013.806,141.113,368.641,-24.367,21.407,-41.460
C07883=1013.807,140.775,368.676,-24.366,21.407,-41.462
C07884=1013.809,140.430,368.711,-24.366,21.407,-41.465
C07885=1013.811,140.036,368.750,-24.365,21.407,-41.469
C07886=1013.812,139.816,368.773,-24.365,21.408,-41.470
C07887=1013.814,139.583,368.797,-24.365,21.408,-41.471
C07888=1013.814,139.342,368.822,-24.365,21.408,-41.473
C07889=1013.816,139.101,368.846,-24.365,21.408,-41.473
C07890=1013.816,138.863,368.871,-24.364,21.408,-41.475
C07891=1013.818,138.635,368.893,-24.364,21.408,-41.477
C07892=1013.820,138.224,368.936,-24.364,21.408,-41.480
C07893=1013.821,137.867,368.972,-24.363,21.408,-41.484
C07894=1013.822,137.527,369.006,-24.363,21.408,-41.486
C07895=1013.824,137.205,369.039,-24.363,21.409,-41.488
C07896=1013.826,136.907,369.069,-24.362,21.409,-41.490
C07897=1013.827,136.631,369.098,-24.362,21.409,-41.491
C07898=1013.828,136.367,369.124,-24.361,21.409,-41.495
C07899=1013.830,136.101,369.151,-24.361,21.410,-41.497
C07900=1013.831,135.823,369.180,-24.361,21.410,-41.499
C07901=1013.832,135.522,369.211,-24.361,21.410,-41.501
C07902=1013.834,135.200,369.243,-24.361,21.411,-41.503
C07903=1013.835,134.866,369.277,-24.360,21.410,-41.506
C07904=1013.837,134.532,369.311,-24.360,21.410,-41.508
C07905=1013.838,134.198,369.344,-24.359,21.411,-41.510
C07906=1013.840,133.864,369.378,-24.359,21.410,-41.513
C07907=1013.842,133.530,369.412,-24.359,21.411,-41.515
C07908=1013.843,133.195,369.447,-24.358,21.411,-41.517
C07909=1013.844,132.862,369.480,-24.358,21.411,-41.521
C07910=1013.846,132.528,369.514,-24.358,21.411,-41.523
C07911=1013.848,132.194,369.548,-24.357,21.412,-41.525
C07912=1013.849,131.859,369.582,-24.357,21.412,-41.528
C07913=1013.850,131.525,369.615,-24.357,21.412,-41.530
C07914=1013.852,131.191,369.649,-24.356,21.412,-41.532
C07915=1013.854,130.857,369.683,-24.356,21.412,-41.535
C07916=1013.856,130.523,369.717,-24.356,21.413,-41.538
C07917=1013.857,130.189,369.750,-24.355,21.413,-41.541
C07918=1013.859,129.855,369.784,-24.355,21.413,-41.543
C07919=1013.860,129.521,369.818,-24.355,21.413,-41.545
C07920=1013.862,129.187,369.851,-24.354,21.414,-41.548
C07921=1013.863,128.853,369.886,-24.354,21.414,-41.550
C07922=1013.865,128.519,369.920,-24.354,21.414,-41.552
C07923=1013.866,128.185,369.953,-24.353,21.414,-41.555
C07924=1013.868,127.851,369.987,-24.353,21.415,-41.558
C07925=1013.870,127.517,370.021,-24.352,21.414,-41.561
C07926=1013.871,127.183,370.054,-24.352,21.415,-41.563
C07927=1013.873,126.849,370.088,-24.352,21.415,-41.565
C07928=1013.874,126.515,370.121,-24.351,21.415,-41.569
C07929=1013.875,126.181,370.155,-24.351,21.415,-41.571
C07930=1013.877,125.847,370.189,-24.351,21.416,-41.572
C07931=1013.878,125.513,370.222,-24.350,21.415,-41.576
C07932=1013.880,125.179,370.256,-24.350,21.416,-41.578
C07933=1013.881,124.845,370.289,-24.349,21.416,-41.581
C07934=1013.883,124.511,370.323,-24.349,21.416,-41.583
C07935=1013.885,124.177,370.355,-24.349,21.416,-41.585
C07936=1013.887,123.843,370.389,-24.348,21.417,-41.589
C07937=1013.888,123.509,370.422,-24.348,21.417,-41.591
C07938=1013.890,123.175,370.456,-24.348,21.417,-41.594
C07939=1013.891,122.841,370.489,-24.347,21.417,-41.596
C07940=1013.893,122.507,370.523,-24.347,21.418,-41.598
C07941=1013.894,122.174,370.557,-24.347,21.418,-41.602
C07942=1013.896,121.840,370.590,-24.346,21.418,-41.604
C07943=1013.897,121.505,370.624,-24.346,21.417,-41.607
C07944=1013.898,121.171,370.658,-24.346,21.418,-41.609
C07945=1013.900,120.837,370.691,-24.345,21.418,-41.613
C07946=1013.902,120.503,370.725,-24.345,21.418,-41.614
C07947=1013.903,120.170,370.758,-24.345,21.419,-41.617
C07948=1013.904,119.836,370.791,-24.344,21.419,-41.620
C07949=1013.906,119.501,370.824,-24.344,21.419,-41.622
C07950=1013.907,119.167,370.858,-24.343,21.419,-41.625
C07951=1013.909,118.833,370.891,-24.343,21.420,-41.628
C07952=1013.910,118.500,370.925,-24.342,21.419,-41.631
C07953=1013.912,118.166,370.958,-24.342,21.420,-41.633
C07954=1013.914,117.832,370.992,-24.342,21.421,-41.635
C07955=1013.915,117.498,371.024,-24.341,21.420,-41.638
C07956=1013.917,117.164,371.058,-24.341,21.421,-41.640
C07957=1013.918,116.830,371.091,-24.341,21.421,-41.644
C07958=1013.919,116.496,371.124,-24.340,21.421,-41.646
C07959=1013.921,116.162,371.158,-24.340,21.421,-41.649
C07960=1013.923,115.829,371.191,-24.340,21.422,-41.652
C07961=1013.924,115.495,371.224,-24.339,21.422,-41.655
C07962=1013.926,115.161,371.257,-24.339,21.422,-41.657
C07963=1013.928,114.827,371.291,-24.338,21.421,-41.660
C07964=1013.929,114.493,371.324,-24.338,21.422,-41.662
C07965=1013.930,114.159,371.356,-24.338,21.423,-41.664
C07966=1013.932,113.825,371.390,-24.337,21.422,-41.668
C07967=1013.933,113.491,371.423,-24.337,21.423,-41.670
C07968=1013.934,113.157,371.457,-24.336,21.423,-41.673
C07969=1013.937,112.823,371.490,-24.336,21.423,-41.675
C07970=1013.938,112.489,371.523,-24.336,21.424,-41.679
C07971=1013.939,112.155,371.556,-24.335,21.424,-41.681
C07972=1013.941,111.821,371.589,-24.335,21.423,-41.684
C07973=1013.942,111.487,371.622,-24.335,21.425,-41.686
C07974=1013.944,111.153,371.656,-24.334,21.424,-41.690
C07975=1013.945,110.819,371.688,-24.334,21.424,-41.692
C07976=1013.946,110.485,371.721,-24.333,21.425,-41.695
C07977=1013.948,110.152,371.754,-24.333,21.425,-41.697
C07978=1013.950,109.818,371.787,-24.333,21.425,-41.701
C07979=1013.952,109.484,371.820,-24.332,21.426,-41.703
C07980=1013.953,109.150,371.854,-24.332,21.425,-41.706
C07981=1013.954,108.816,371.886,-24.332,21.426,-41.708
C07982=1013.955,108.482,371.919,-24.331,21.426,-41.712
C07983=1013.957,108.148,371.952,-24.331,21.426,-41.714
C07984=1013.959,107.814,371.986,-24.330,21.427,-41.718
C07985=1013.960,107.479,372.018,-24.330,21.427,-41.719
C07986=1013.961,107.146,372.051,-24.329,21.427,-41.723
C07987=1013.963,106.812,372.085,-24.329,21.428,-41.725
C07988=1013.964,106.478,372.117,-24.329,21.427,-41.728
C07989=1013.965,106.144,372.150,-24.328,21.427,-41.730
C07990=1013.967,105.809,372.183,-24.328,21.428,-41.734
C07991=1013.968,105.476,372.216,-24.328,21.428,-41.736
C07992=1013.971,105.142,372.249,-24.327,21.428,-41.739
C07993=1013.972,104.808,372.282,-24.327,21.429,-41.742
C07994=1013.973,104.474,372.315,-24.326,21.428,-41.745
C07995=1013.975,104.139,372.347,-24.326,21.430,-41.747
C07996=1013.976,103.806,372.380,-24.326,21.429,-41.751
C07997=1013.978,103.471,372.413,-24.325,21.429,-41.752
C07998=1013.979,103.138,372.446,-24.325,21.430,-41.756
C07999=1013.980,102.803,372.479,-24.324,21.429,-41.760
C08000=1013.981,102.470,372.512,-24.324,21.431,-41.762
C08001=1013.983,102.135,372.544,-24.324,21.430,-41.765
C08002=1013.984,101.801,372.577,-24.323,21.430,-41.767
C08003=1013.986,101.467,372.610,-24.323,21.431,-41.771
C08004=1013.987,101.133,372.643,-24.323,21.431,-41.773
C08005=1013.989,100.798,372.675,-24.322,21.431,-41.776
C08006=1013.990,100.465,372.708,-24.322,21.432,-41.778
C08007=1013.991,100.130,372.741,-24.321,21.431,-41.782
C08008=1013.993,99.796,372.773,-24.321,21.432,-41.785
C08009=1013.994,99.462,372.806,-24.320,21.432,-41.787
C08010=1013.995,99.128,372.839,-24.320,21.432,-41.791
C08011=1013.997,98.794,372.871,-24.320,21.433,-41.793
C08012=1013.998,98.459,372.904,-24.319,21.432,-41.796
C08013=1013.999,98.126,372.937,-24.319,21.433,-41.799
C08014=1014.001,97.791,372.970,-24.318,21.433,-41.802
C08015=1014.002,97.457,373.002,-24.318,21.433,-41.806
C08016=1014.004,97.123,373.035,-24.318,21.434,-41.808
C08017=1014.005,96.789,373.068,-24.317,21.434,-41.811
C08018=1014.007,96.454,373.100,-24.317,21.434,-41.813
C08019=1014.008,96.120,373.133,-24.316,21.434,-41.817
C08020=1014.010,95.786,373.165,-24.316,21.435,-41.819
C08021=1014.011,95.451,373.198,-24.316,21.435,-41.822
C08022=1014.013,95.117,373.230,-24.315,21.435,-41.826
C08023=1014.014,94.783,373.263,-24.315,21.435,-41.828
C08024=1014.015,94.449,373.295,-24.314,21.436,-41.832
C08025=1014.016,94.115,373.328,-24.314,21.436,-41.833
C08026=1014.017,93.781,373.361,-24.314,21.436,-41.837
C08027=1014.019,93.446,373.393,-24.313,21.436,-41.841
C08028=1014.020,93.112,373.426,-24.313,21.436,-41.842
C08029=1014.022,92.778,373.458,-24.312,21.437,-41.846
C08030=1014.023,92.443,373.491,-24.312,21.436,-41.849
C08031=1014.025,92.109,373.523,-24.311,21.437,-41.852
C08032=1014.026,91.775,373.556,-24.311,21.437,-41.855
C08033=1014.027,91.441,373.588,-24.311,21.438,-41.857
C08034=1014.029,91.106,373.620,-24.310,21.438,-41.861
C08035=1014.030,90.771,373.652,-24.310,21.438,-41.865
C08036=1014.031,90.436,373.685,-24.309,21.438,-41.866
C08037=1014.033,90.102,373.717,-24.309,21.439,-41.870
C08038=1014.034,89.767,373.750,-24.308,21.438,-41.874
C08039=1014.035,89.435,373.782,-24.308,21.440,-41.876
C08040=1014.037,89.106,373.814,-24.308,21.439,-41.879
C08041=1014.038,88.781,373.845,-24.307,21.439,-41.881
C08042=1014.040,88.460,373.876,-24.307,21.440,-41.885
C08043=1014.040,88.139,373.907,-24.306,21.439,-41.888
C08044=1014.042,87.817,373.939,-24.306,21.441,-41.890
C08045=1014.043,87.491,373.970,-24.305,21.440,-41.894
C08046=1014.044,87.158,374.002,-24.305,21.441,-41.898
C08047=1014.045,86.821,374.034,-24.305,21.441,-41.899
C08048=1014.048,86.482,374.067,-24.304,21.441,-41.903
C08049=1014.048,86.141,374.100,-24.304,21.441,-41.906
C08050=1014.049,85.799,374.133,-24.303,21.442,-41.909
C08051=1014.051,85.456,374.165,-24.303,21.442,-41.912
C08052=1014.052,85.112,374.200,-24.302,21.442,-41.916
C08053=1014.053,84.766,374.232,-24.302,21.443,-41.918
C08054=1014.055,84.420,374.266,-24.302,21.443,-41.922
C08055=1014.056,84.072,374.299,-24.301,21.443,-41.925
C08056=1014.058,83.723,374.333,-24.301,21.443,-41.929
C08057=1014.059,83.373,374.366,-24.300,21.444,-41.931
C08058=1014.060,83.022,374.400,-24.300,21.444,-41.935
C08059=1014.061,82.670,374.434,-24.299,21.444,-41.938
C08060=1014.063,82.317,374.468,-24.299,21.444,-41.942
C08061=1014.065,81.964,374.502,-24.298,21.444,-41.945
C08062=1014.066,81.609,374.536,-24.298,21.445,-41.947
C08063=1014.067,81.253,374.569,-24.298,21.446,-41.951
C08064=1014.068,80.898,374.604,-24.297,21.445,-41.955
C08065=1014.070,80.541,374.638,-24.297,21.446,-41.958
C08066=1014.071,80.185,374.673,-24.296,21.446,-41.962
C08067=1014.072,79.830,374.706,-24.296,21.446,-41.964
C08068=1014.074,79.479,374.740,-24.295,21.447,-41.968
C08069=1014.075,79.134,374.773,-24.295,21.446,-41.971
C08070=1014.076,78.795,374.805,-24.295,21.448,-41.973
C08071=1014.078,78.462,374.836,-24.294,21.447,-41.977
C08072=1014.078,78.134,374.868,-24.293,21.448,-41.980
C08073=1014.080,77.810,374.899,-24.293,21.448,-41.984
C08074=1014.081,77.486,374.930,-24.292,21.448,-41.987
C08075=1014.082,77.162,374.961,-24.292,21.449,-41.990
C08076=1014.083,76.836,374.992,-24.292,21.449,-41.994
C08077=1014.084,76.506,375.023,-24.291,21.449,-41.997
C08078=1014.086,76.170,375.055,-24.291,21.449,-42.001
C08079=1014.087,75.828,375.088,-24.290,21.449,-42.004
C08080=1014.088,75.479,375.121,-24.290,21.450,-42.006
C08081=1014.090,75.125,375.155,-24.289,21.450,-42.010
C08082=1014.091,74.768,375.189,-24.289,21.450,-42.013
C08083=1014.092,74.410,375.222,-24.288,21.451,-42.017
C08084=1014.094,74.053,375.257,-24.288,21.451,-42.019
C08085=1014.095,73.698,375.290,-24.288,21.451,-42.023
C08086=1014.096,73.345,375.323,-24.287,21.452,-42.027
C08087=1014.097,72.993,375.357,-24.286,21.451,-42.030
C08088=1014.098,72.644,375.390,-24.286,21.452,-42.034
C08089=1014.100,72.296,375.424,-24.285,21.452,-42.037
C08090=1014.101,71.950,375.456,-24.285,21.453,-42.041
C08091=1014.102,71.604,375.489,-24.285,21.453,-42.043
C08092=1014.103,71.259,375.522,-24.284,21.453,-42.047
C08093=1014.105,70.914,375.554,-24.284,21.454,-42.051
C08094=1014.106,70.570,375.587,-24.283,21.453,-42.054
C08095=1014.107,70.226,375.619,-24.283,21.454,-42.058
C08096=1014.108,69.882,375.652,-24.282,21.454,-42.061
C08097=1014.109,69.537,375.685,-24.282,21.455,-42.063
C08098=1014.110,69.193,375.717,-24.281,21.455,-42.067
C08099=1014.112,68.850,375.749,-24.281,21.456,-42.071
C08100=1014.112,68.507,375.781,-24.280,21.455,-42.074
C08101=1014.114,68.166,375.814,-24.280,21.456,-42.078
C08102=1014.115,67.826,375.846,-24.279,21.456,-42.082
C08103=1014.115,67.487,375.878,-24.279,21.456,-42.085
C08104=1014.117,67.149,375.910,-24.279,21.457,-42.087
C08105=1014.118,66.811,375.941,-24.278,21.457,-42.091
C08106=1014.120,66.474,375.973,-24.278,21.457,-42.094
C08107=1014.121,66.139,376.005,-24.277,21.457,-42.098
C08108=1014.121,65.806,376.036,-24.277,21.458,-42.102
C08109=1014.123,65.467,376.068,-24.276,21.457,-42.105
C08110=1014.124,65.112,376.101,-24.276,21.459,-42.108
C08111=1014.126,64.735,376.136,-24.275,21.458,-42.113
C08112=1014.127,64.339,376.174,-24.274,21.459,-42.116
C08113=1014.128,63.954,376.210,-24.274,21.459,-42.120
C08114=1014.129,63.597,376.243,-24.274,21.460,-42.124
C08115=1014.137,63.225,376.274,-24.273,21.460,-42.128
C08116=1014.141,63.006,376.292,-24.273,21.461,-42.130
C08117=1014.145,62.783,376.311,-24.272,21.460,-42.131
C08118=1014.153,62.387,376.344,-24.272,21.460,-42.135
C08119=1014.160,62.051,376.372,-24.271,21.461,-42.139
C08120=1014.166,61.716,376.400,-24.271,21.461,-42.142
C08121=1014.172,61.381,376.428,-24.270,21.462,-42.146
C08122=1014.178,61.046,376.457,-24.270,21.461,-42.149
C08123=1014.185,60.712,376.484,-24.269,21.462,-42.153
C08124=1014.192,60.376,376.513,-24.269,21.462,-42.157
C08125=1014.198,60.041,376.541,-24.268,21.462,-42.160
C08126=1014.204,59.707,376.569,-24.268,21.463,-42.163
C08127=1014.210,59.372,376.597,-24.268,21.464,-42.166
C08128=1014.216,59.037,376.625,-24.267,21.464,-42.170
C08129=1014.222,58.702,376.653,-24.267,21.464,-42.173
C08130=1014.228,58.367,376.681,-24.266,21.464,-42.177
C08131=1014.234,58.032,376.709,-24.266,21.465,-42.181
C08132=1014.240,57.697,376.737,-24.265,21.464,-42.184
C08133=1014.246,57.362,376.765,-24.264,21.465,-42.188
C08134=1014.253,57.027,376.793,-24.264,21.465,-42.192
C08135=1014.259,56.692,376.821,-24.264,21.466,-42.194
C08136=1014.265,56.357,376.849,-24.263,21.466,-42.197
C08137=1014.271,56.022,376.877,-24.263,21.466,-42.201
C08138=1014.276,55.688,376.905,-24.262,21.467,-42.205
C08139=1014.282,55.353,376.933,-24.262,21.467,-42.209
C08140=1014.288,55.018,376.961,-24.261,21.467,-42.212
C08141=1014.295,54.684,376.989,-24.261,21.467,-42.216
C08142=1014.300,54.349,377.017,-24.260,21.468,-42.220
C08143=1014.306,54.014,377.045,-24.260,21.468,-42.223
C08144=1014.312,53.678,377.073,-24.259,21.468,-42.227
C08145=1014.317,53.344,377.101,-24.259,21.468,-42.230
C08146=1014.323,53.009,377.130,-24.258,21.469,-42.234
C08147=1014.329,52.674,377.158,-24.258,21.469,-42.238
C08148=1014.335,52.340,377.185,-24.257,21.470,-42.240
C08149=1014.340,52.004,377.213,-24.257,21.470,-42.244
C08150=1014.346,51.669,377.241,-24.256,21.470,-42.247
C08151=1014.352,51.334,377.269,-24.256,21.471,-42.251
C08152=1014.357,51.000,377.297,-24.255,21.471,-42.254
C08153=1014.362,50.665,377.326,-24.255,21.471,-42.258
C08154=1014.368,50.330,377.353,-24.254,21.471,-42.262
C08155=1014.374,49.995,377.381,-24.254,21.472,-42.266
C08156=1014.378,49.660,377.410,-24.253,21.472,-42.269
C08157=1014.385,49.326,377.438,-24.253,21.472,-42.273
C08158=1014.390,48.991,377.465,-24.252,21.473,-42.277
C08159=1014.395,48.656,377.493,-24.252,21.473,-42.280
C08160=1014.401,48.321,377.522,-24.251,21.473,-42.284
C08161=1014.406,47.987,377.549,-24.251,21.473,-42.287
C08162=1014.411,47.651,377.577,-24.250,21.474,-42.291
C08163=1014.417,47.316,377.605,-24.250,21.474,-42.295
C08164=1014.422,46.982,377.634,-24.249,21.475,-42.299
C08165=1014.427,46.647,377.661,-24.249,21.475,-42.302
C08166=1014.432,46.312,377.689,-24.248,21.475,-42.306
C08167=1014.438,45.977,377.718,-24.248,21.475,-42.309
C08168=1014.443,45.643,377.745,-24.247,21.476,-42.313
C08169=1014.448,45.307,377.773,-24.247,21.476,-42.317
C08170=1014.453,44.973,377.801,-24.246,21.477,-42.321
C08171=1014.458,44.638,377.829,-24.246,21.477,-42.325
C08172=1014.463,44.303,377.856,-24.245,21.477,-42.328
C08173=1014.468,43.969,377.885,-24.245,21.477,-42.332
C08174=1014.473,43.634,377.912,-24.244,21.478,-42.335
C08175=1014.478,43.299,377.940,-24.244,21.478,-42.339
C08176=1014.483,42.965,377.968,-24.243,21.479,-42.343
C08177=1014.488,42.629,377.996,-24.243,21.479,-42.347
C08178=1014.493,42.294,378.025,-24.242,21.479,-42.350
C08179=1014.498,41.960,378.052,-24.242,21.479,-42.354
C08180=1014.502,41.625,378.081,-24.241,21.480,-42.357
C08181=1014.508,41.290,378.108,-24.241,21.480,-42.361
C08182=1014.513,40.955,378.136,-24.240,21.481,-42.365
C08183=1014.518,40.621,378.164,-24.240,21.481,-42.369
C08184=1014.523,40.286,378.192,-24.239,21.481,-42.372
C08185=1014.527,39.951,378.221,-24.239,21.481,-42.376
C08186=1014.532,39.617,378.248,-24.238,21.482,-42.380
C08187=1014.536,39.282,378.276,-24.238,21.482,-42.383
C08188=1014.542,38.947,378.304,-24.237,21.483,-42.387
C08189=1014.546,38.613,378.332,-24.237,21.483,-42.391
C08190=1014.550,38.278,378.359,-24.236,21.483,-42.395
C08191=1014.555,37.944,378.387,-24.236,21.483,-42.398
C08192=1014.560,37.608,378.415,-24.235,21.484,-42.402
C08193=1014.565,37.274,378.444,-24.235,21.484,-42.405
C08194=1014.570,36.939,378.471,-24.234,21.485,-42.409
C08195=1014.574,36.605,378.499,-24.234,21.485,-42.413
C08196=1014.578,36.270,378.527,-24.233,21.485,-42.418
C08197=1014.583,35.935,378.555,-24.232,21.485,-42.422
C08198=1014.587,35.601,378.583,-24.232,21.486,-42.426
C08199=1014.592,35.266,378.610,-24.231,21.485,-42.429
C08200=1014.596,34.932,378.638,-24.231,21.486,-42.433
C08201=1014.601,34.597,378.667,-24.230,21.486,-42.437
C08202=1014.605,34.262,378.694,-24.230,21.487,-42.440
C08203=1014.610,33.928,378.722,-24.229,21.487,-42.444
C08204=1014.614,33.593,378.749,-24.229,21.488,-42.448
C08205=1014.618,33.259,378.778,-24.228,21.488,-42.452
C08206=1014.622,32.924,378.806,-24.228,21.489,-42.455
C08207=1014.627,32.590,378.833,-24.227,21.489,-42.459
C08208=1014.631,32.255,378.861,-24.226,21.489,-42.464
C08209=1014.635,31.921,378.889,-24.226,21.489,-42.468
C08210=1014.640,31.586,378.916,-24.225,21.489,-42.471
C08211=1014.644,31.252,378.944,-24.225,21.490,-42.475
C08212=1014.648,30.917,378.972,-24.224,21.490,-42.479
C08213=1014.652,30.583,379.000,-24.224,21.491,-42.483
C08214=1014.657,30.248,379.027,-24.223,21.491,-42.486
C08215=1014.660,29.914,379.055,-24.223,21.492,-42.490
C08216=1014.664,29.580,379.083,-24.222,21.492,-42.494
C08217=1014.669,29.246,379.111,-24.222,21.493,-42.498
C08218=1014.673,28.911,379.138,-24.221,21.492,-42.503
C08219=1014.676,28.577,379.166,-24.221,21.493,-42.507
C08220=1014.680,28.242,379.194,-24.220,21.493,-42.510
C08221=1014.685,27.908,379.221,-24.220,21.494,-42.514
C08222=1014.688,27.574,379.249,-24.219,21.494,-42.518
C08223=1014.692,27.239,379.277,-24.219,21.495,-42.522
C08224=1014.696,26.905,379.305,-24.218,21.494,-42.525
C08225=1014.701,26.571,379.332,-24.217,21.494,-42.530
C08226=1014.704,26.237,379.360,-24.217,21.495,-42.534
C08227=1014.708,25.902,379.388,-24.216,21.495,-42.538
C08228=1014.712,25.568,379.416,-24.216,21.496,-42.541
C08229=1014.716,25.234,379.444,-24.215,21.496,-42.545
C08230=1014.719,24.900,379.471,-24.215,21.497,-42.549
C08231=1014.723,24.565,379.498,-24.214,21.497,-42.553
C08232=1014.727,24.230,379.526,-24.213,21.497,-42.558
C08233=1014.731,23.904,379.554,-24.213,21.498,-42.560
C08234=1014.735,23.610,379.577,-24.213,21.498,-42.562
C08235=1014.738,23.358,379.598,-24.212,21.498,-42.565
C08236=1014.742,22.950,379.632,-24.211,21.499,-42.573
C08237=1014.746,22.540,379.666,-24.210,21.499,-42.580
C08238=1014.749,22.288,379.686,-24.210,21.500,-42.582
C08239=1014.752,21.993,379.711,-24.210,21.501,-42.584
C08240=1014.755,21.670,379.738,-24.209,21.500,-42.588
C08241=1014.759,21.314,379.767,-24.209,21.501,-42.593
C08242=1014.762,21.106,379.785,-24.208,21.501,-42.597
C08243=1014.764,20.879,379.803,-24.208,21.502,-42.599
C08244=1014.766,20.637,379.823,-24.208,21.502,-42.601
C08245=1014.769,20.389,379.844,-24.207,21.502,-42.603
C08246=1014.772,20.142,379.864,-24.207,21.502,-42.604
C08247=1014.775,19.907,379.884,-24.207,21.502,-42.608
C08248=1014.778,19.489,379.918,-24.206,21.503,-42.613
C08249=1014.783,19.141,379.946,-24.205,21.502,-42.619
C08250=1014.785,18.809,379.973,-24.205,21.503,-42.622
C08251=1014.789,18.477,380.001,-24.204,21.503,-42.626
C08252=1014.792,18.146,380.028,-24.204,21.504,-42.630
C08253=1014.796,17.815,380.055,-24.203,21.504,-42.634
C08254=1014.799,17.485,380.082,-24.202,21.504,-42.639
C08255=1014.802,17.155,380.110,-24.202,21.505,-42.643
C08256=1014.805,16.826,380.137,-24.201,21.505,-42.646
C08257=1014.808,16.498,380.164,-24.201,21.506,-42.650
C08258=1014.813,16.169,380.191,-24.200,21.506,-42.654
C08259=1014.815,15.842,380.217,-24.200,21.507,-42.658
C08260=1014.819,15.515,380.245,-24.199,21.507,-42.663
C08261=1014.822,15.189,380.272,-24.199,21.507,-42.667
C08262=1014.825,14.863,380.298,-24.198,21.508,-42.670
C08263=1014.828,14.537,380.325,-24.198,21.508,-42.674
C08264=1014.831,14.213,380.352,-24.197,21.509,-42.678
C08265=1014.834,13.888,380.379,-24.197,21.509,-42.682
C08266=1014.837,13.564,380.405,-24.196,21.509,-42.687
C08267=1014.840,13.240,380.431,-24.195,21.509,-42.691
C08268=1014.843,12.915,380.458,-24.195,21.510,-42.694
C08269=1014.846,12.592,380.485,-24.194,21.510,-42.698
C08270=1014.849,12.268,380.511,-24.194,21.511,-42.702
C08271=1014.852,11.946,380.538,-24.193,21.511,-42.707
C08272=1014.854,11.622,380.565,-24.193,21.511,-42.711
C08273=1014.857,11.298,380.591,-24.192,21.512,-42.715
C08274=1014.861,10.976,380.618,-24.192,21.512,-42.718
C08275=1014.864,10.655,380.643,-24.191,21.513,-42.722
C08276=1014.866,10.336,380.670,-24.191,21.513,-42.726
C08277=1014.869,10.020,380.695,-24.190,21.514,-42.730
C08278=1014.871,9.704,380.721,-24.190,21.514,-42.733
C08279=1014.875,9.390,380.747,-24.189,21.514,-42.738
C08280=1014.878,9.075,380.773,-24.188,21.515,-42.742
C08281=1014.880,8.760,380.799,-24.188,21.515,-42.746
C08282=1014.883,8.444,380.824,-24.187,21.516,-42.750
C08283=1014.885,8.125,380.851,-24.186,21.515,-42.755
C08284=1014.888,7.805,380.876,-24.186,21.516,-42.759
C08285=1014.891,7.482,380.903,-24.186,21.516,-42.762
C08286=1014.893,7.156,380.930,-24.185,21.517,-42.766
C08287=1014.896,6.829,380.956,-24.185,21.517,-42.770
C08288=1014.899,6.500,380.983,-24.184,21.518,-42.774
C08289=1014.901,6.172,381.009,-24.183,21.518,-42.779
C08290=1014.904,5.842,381.037,-24.183,21.518,-42.783
C08291=1014.906,5.512,381.063,-24.182,21.519,-42.786
C08292=1014.910,5.182,381.090,-24.181,21.518,-42.792
C08293=1014.912,4.851,381.117,-24.181,21.519,-42.795
C08294=1014.915,4.520,381.145,-24.180,21.519,-42.799
C08295=1014.917,4.188,381.172,-24.180,21.521,-42.803
C08296=1014.920,3.859,381.198,-24.179,21.520,-42.807
C08297=1014.922,3.546,381.224,-24.179,21.521,-42.810
C08298=1014.925,3.257,381.247,-24.179,21.521,-42.814
C08299=1014.926,2.987,381.269,-24.178,21.522,-42.818
C08300=1014.928,2.725,381.290,-24.177,21.522,-42.823
C08301=1014.931,2.456,381.312,-24.177,21.522,-42.827
C08302=1014.933,2.169,381.336,-24.176,21.523,-42.831
C08303=1014.935,1.855,381.361,-24.176,21.523,-42.834
C08304=1014.938,1.525,381.388,-24.175,21.523,-42.838
C08305=1014.940,1.192,381.415,-24.175,21.524,-42.842
C08306=1014.942,0.858,381.442,-24.174,21.525,-42.846
C08307=1014.945,0.523,381.469,-24.173,21.525,-42.851
C08308=1014.947,0.187,381.496,-24.173,21.525,-42.855
C08309=1014.949,-0.149,381.524,-24.172,21.526,-42.858
C08310=1014.951,-0.488,381.551,-24.172,21.526,-42.864
C08311=1014.954,-0.829,381.579,-24.171,21.526,-42.867
C08312=1014.957,-1.170,381.606,-24.170,21.527,-42.873
C08313=1014.958,-1.514,381.634,-24.170,21.527,-42.877
C08314=1014.961,-1.858,381.662,-24.169,21.528,-42.880
C08315=1014.963,-2.205,381.690,-24.169,21.528,-42.886
C08316=1014.966,-2.553,381.718,-24.168,21.529,-42.890
C08317=1014.968,-2.903,381.747,-24.167,21.529,-42.895
C08318=1014.970,-3.254,381.775,-24.167,21.529,-42.899
C08319=1014.973,-3.607,381.803,-24.166,21.529,-42.904
C08320=1014.975,-3.961,381.832,-24.166,21.531,-42.908
C08321=1014.977,-4.318,381.861,-24.165,21.530,-42.913
C08322=1014.979,-4.680,381.890,-24.164,21.531,-42.919
C08323=1014.982,-5.046,381.920,-24.164,21.532,-42.923
C08324=1014.984,-5.416,381.950,-24.163,21.532,-42.928
C08325=1014.986,-5.791,381.980,-24.163,21.533,-42.932
C08326=1014.988,-6.166,382.010,-24.162,21.533,-42.937
C08327=1014.990,-6.541,382.040,-24.161,21.533,-42.941
C08328=1014.993,-6.916,382.071,-24.160,21.534,-42.947
C08329=1014.996,-7.287,382.100,-24.160,21.534,-42.952
C08330=1014.997,-7.655,382.130,-24.159,21.535,-42.956
C08331=1015.000,-8.022,382.159,-24.158,21.535,-42.961
C08332=1015.001,-8.386,382.189,-24.158,21.536,-42.967
C08333=1015.003,-8.748,382.218,-24.157,21.536,-42.971
C08334=1015.005,-9.111,382.247,-24.156,21.536,-42.976
C08335=1015.008,-9.474,382.276,-24.156,21.537,-42.982
C08336=1015.009,-9.836,382.305,-24.155,21.538,-42.985
C08337=1015.012,-10.197,382.334,-24.154,21.538,-42.991
C08338=1015.013,-10.558,382.363,-24.154,21.539,-42.995
C08339=1015.015,-10.917,382.392,-24.153,21.539,-43.000
C08340=1015.017,-11.277,382.420,-24.152,21.539,-43.006
C08341=1015.019,-11.634,382.449,-24.152,21.540,-43.009
C08342=1015.021,-11.991,382.477,-24.151,21.540,-43.014
C08343=1015.023,-12.346,382.506,-24.151,21.541,-43.019
C08344=1015.024,-12.699,382.534,-24.150,21.541,-43.024
C08345=1015.025,-13.051,382.563,-24.149,21.542,-43.028
C08346=1015.028,-13.401,382.591,-24.149,21.542,-43.033
C08347=1015.029,-13.751,382.619,-24.148,21.543,-43.037
C08348=1015.031,-14.096,382.646,-24.147,21.543,-43.042
C08349=1015.033,-14.440,382.674,-24.147,21.544,-43.046
C08350=1015.034,-14.782,382.701,-24.146,21.544,-43.052
C08351=1015.035,-15.122,382.728,-24.146,21.544,-43.055
C08352=1015.038,-15.460,382.755,-24.145,21.545,-43.061
C08353=1015.038,-15.797,382.782,-24.145,21.546,-43.065
C08354=1015.040,-16.132,382.808,-24.144,21.546,-43.070
C08355=1015.042,-16.467,382.835,-24.143,21.546,-43.074
C08356=1015.044,-16.800,382.862,-24.142,21.547,-43.079
C08357=1015.044,-17.134,382.889,-24.142,21.547,-43.083
C08358=1015.046,-17.467,382.915,-24.141,21.547,-43.088
C08359=1015.048,-17.799,382.942,-24.141,21.548,-43.092
C08360=1015.048,-18.164,382.970,-24.140,21.549,-43.100
C08361=1015.050,-18.387,382.988,-24.139,21.548,-43.103
C08362=1015.051,-18.633,383.008,-24.139,21.549,-43.105
C08363=1015.052,-18.895,383.028,-24.139,21.550,-43.107
C08364=1015.053,-19.157,383.050,-24.139,21.550,-43.109
C08365=1015.053,-19.405,383.069,-24.138,21.550,-43.112
C08366=1015.055,-19.821,383.103,-24.137,21.550,-43.118
C08367=1015.056,-19.994,383.116,-24.137,21.551,-43.122
C08368=1015.057,-20.326,383.142,-24.136,21.551,-43.127
C08369=1015.058,-20.659,383.169,-24.136,21.552,-43.131
C08370=1015.060,-20.992,383.195,-24.135,21.553,-43.135
C08371=1015.061,-21.324,383.221,-24.134,21.552,-43.140
C08372=1015.062,-21.657,383.248,-24.134,21.553,-43.144
C08373=1015.063,-21.991,383.274,-24.133,21.554,-43.149
C08374=1015.064,-22.323,383.300,-24.133,21.554,-43.153
C08375=1015.066,-22.655,383.327,-24.132,21.554,-43.158
C08376=1015.067,-22.989,383.353,-24.131,21.556,-43.162
C08377=1015.068,-23.321,383.379,-24.131,21.555,-43.168
C08378=1015.068,-23.654,383.406,-24.130,21.556,-43.171
C08379=1015.070,-23.987,383.432,-24.129,21.556,-43.177
C08380=1015.070,-24.320,383.458,-24.129,21.557,-43.181
C08381=1015.072,-24.652,383.485,-24.128,21.557,-43.186
C08382=1015.073,-24.985,383.510,-24.128,21.558,-43.190
C08383=1015.074,-25.318,383.537,-24.127,21.558,-43.195
C08384=1015.075,-25.650,383.563,-24.126,21.559,-43.199
C08385=1015.076,-25.984,383.589,-24.126,21.559,-43.204
C08386=1015.077,-26.316,383.616,-24.125,21.559,-43.208
C08387=1015.077,-26.649,383.642,-24.124,21.560,-43.214
C08388=1015.078,-26.982,383.668,-24.124,21.560,-43.217
C08389=1015.079,-27.315,383.695,-24.123,21.560,-43.223
C08390=1015.080,-27.647,383.721,-24.123,21.562,-43.227
C08391=1015.081,-27.980,383.746,-24.122,21.562,-43.232
C08392=1015.082,-28.312,383.772,-24.121,21.562,-43.236
C08393=1015.082,-28.645,383.799,-24.120,21.562,-43.241
C08394=1015.084,-28.978,383.825,-24.120,21.563,-43.245
C08395=1015.084,-29.311,383.851,-24.119,21.563,-43.250
C08396=1015.085,-29.643,383.877,-24.119,21.564,-43.254
C08397=1015.086,-29.977,383.903,-24.118,21.565,-43.260
C08398=1015.086,-30.309,383.929,-24.118,21.565,-43.264
C08399=1015.087,-30.642,383.956,-24.117,21.565,-43.269
C08400=1015.088,-30.975,383.981,-24.116,21.566,-43.273
C08401=1015.088,-31.307,384.007,-24.116,21.566,-43.278
C08402=1015.089,-31.640,384.034,-24.115,21.567,-43.282
C08403=1015.089,-31.973,384.059,-24.114,21.567,-43.287
C08404=1015.090,-32.305,384.086,-24.114,21.568,-43.291
C08405=1015.090,-32.638,384.112,-24.113,21.568,-43.296
C08406=1015.091,-32.971,384.137,-24.113,21.569,-43.301
C08407=1015.092,-33.304,384.164,-24.112,21.569,-43.306
C08408=1015.092,-33.636,384.190,-24.111,21.570,-43.310
C08409=1015.093,-33.969,384.216,-24.111,21.570,-43.315
C08410=1015.094,-34.302,384.242,-24.110,21.571,-43.319
C08411=1015.094,-34.634,384.268,-24.109,21.571,-43.324
C08412=1015.094,-34.967,384.293,-24.109,21.572,-43.328
C08413=1015.095,-35.300,384.319,-24.108,21.572,-43.334
C08414=1015.095,-35.632,384.346,-24.108,21.573,-43.337
C08415=1015.096,-35.965,384.371,-24.107,21.573,-43.343
C08416=1015.096,-36.297,384.397,-24.107,21.574,-43.347
C08417=1015.097,-36.631,384.422,-24.106,21.574,-43.352
C08418=1015.097,-36.963,384.449,-24.105,21.574,-43.357
C08419=1015.097,-37.295,384.474,-24.105,21.575,-43.361
C08420=1015.098,-37.628,384.500,-24.104,21.575,-43.366
C08421=1015.098,-37.961,384.526,-24.103,21.576,-43.371
C08422=1015.097,-38.294,384.552,-24.102,21.576,-43.376
C08423=1015.098,-38.627,384.578,-24.102,21.577,-43.380
C08424=1015.098,-38.959,384.604,-24.101,21.577,-43.385
C08425=1015.099,-39.292,384.630,-24.101,21.578,-43.389
C08426=1015.099,-39.625,384.655,-24.100,21.578,-43.394
C08427=1015.099,-39.957,384.681,-24.100,21.579,-43.398
C08428=1015.099,-40.289,384.707,-24.099,21.579,-43.404
C08429=1015.100,-40.622,384.732,-24.098,21.580,-43.409
C08430=1015.099,-40.955,384.758,-24.098,21.580,-43.413
C08431=1015.100,-41.287,384.784,-24.097,21.580,-43.418
C08432=1015.100,-41.620,384.809,-24.096,21.582,-43.422
C08433=1015.100,-41.952,384.835,-24.096,21.582,-43.427
C08434=1015.100,-42.285,384.862,-24.095,21.582,-43.431
C08435=1015.100,-42.618,384.887,-24.094,21.583,-43.437
C08436=1015.100,-42.950,384.912,-24.094,21.583,-43.442
C08437=1015.100,-43.283,384.939,-24.093,21.583,-43.446
C08438=1015.100,-43.616,384.964,-24.092,21.584,-43.451
C08439=1015.100,-43.948,384.989,-24.092,21.585,-43.455
C08440=1015.100,-44.280,385.015,-24.091,21.585,-43.461
C08441=1015.100,-44.613,385.040,-24.091,21.586,-43.465
C08442=1015.100,-44.946,385.067,-24.090,21.586,-43.470
C08443=1015.099,-45.278,385.092,-24.089,21.586,-43.475
C08444=1015.100,-45.611,385.117,-24.089,21.587,-43.479
C08445=1015.099,-45.943,385.143,-24.088,21.588,-43.485
C08446=1015.099,-46.276,385.169,-24.088,21.588,-43.488
C08447=1015.099,-46.608,385.194,-24.087,21.588,-43.494
C08448=1015.099,-46.941,385.219,-24.086,21.590,-43.498
C08449=1015.099,-47.273,385.245,-24.086,21.589,-43.503
C08450=1015.098,-47.606,385.270,-24.085,21.589,-43.508
C08451=1015.098,-47.939,385.296,-24.084,21.591,-43.512
C08452=1015.098,-48.271,385.322,-24.083,21.591,-43.518
C08453=1015.098,-48.604,385.347,-24.083,21.592,-43.522
C08454=1015.098,-48.936,385.372,-24.082,21.592,-43.527
C08455=1015.097,-49.268,385.398,-24.081,21.592,-43.532
C08456=1015.097,-49.602,385.423,-24.081,21.593,-43.536
C08457=1015.096,-49.933,385.448,-24.080,21.593,-43.542
C08458=1015.096,-50.266,385.474,-24.080,21.595,-43.546
C08459=1015.096,-50.598,385.499,-24.079,21.594,-43.551
C08460=1015.095,-50.931,385.525,-24.079,21.595,-43.555
C08461=1015.095,-51.263,385.550,-24.078,21.596,-43.560
C08462=1015.094,-51.595,385.576,-24.077,21.596,-43.566
C08463=1015.094,-51.928,385.601,-24.077,21.597,-43.570
C08464=1015.093,-52.260,385.626,-24.076,21.597,-43.575
C08465=1015.093,-52.592,385.652,-24.075,21.597,-43.579
C08466=1015.092,-52.925,385.677,-24.075,21.598,-43.584
C08467=1015.092,-53.257,385.702,-24.074,21.598,-43.589
C08468=1015.091,-53.589,385.728,-24.074,21.600,-43.594
C08469=1015.090,-53.921,385.753,-24.073,21.599,-43.599
C08470=1015.090,-54.253,385.778,-24.072,21.600,-43.603
C08471=1015.090,-54.586,385.803,-24.072,21.601,-43.608
C08472=1015.089,-54.919,385.829,-24.071,21.601,-43.613
C08473=1015.088,-55.251,385.854,-24.070,21.602,-43.618
C08474=1015.088,-55.583,385.879,-24.070,21.602,-43.623
C08475=1015.086,-55.916,385.904,-24.069,21.603,-43.627
C08476=1015.086,-56.249,385.929,-24.068,21.603,-43.632
C08477=1015.085,-56.581,385.955,-24.068,21.603,-43.637
C08478=1015.084,-56.915,385.980,-24.067,21.605,-43.642
C08479=1015.084,-57.249,386.005,-24.066,21.604,-43.647
C08480=1015.083,-57.582,386.030,-24.066,21.605,-43.652
C08481=1015.082,-57.915,386.055,-24.065,21.606,-43.656
C08482=1015.081,-58.250,386.080,-24.064,21.606,-43.662
C08483=1015.080,-58.584,386.106,-24.064,21.607,-43.666
C08484=1015.080,-58.920,386.132,-24.063,21.607,-43.671
C08485=1015.079,-59.255,386.157,-24.062,21.608,-43.676
C08486=1015.078,-59.590,386.182,-24.062,21.608,-43.680
C08487=1015.077,-59.927,386.207,-24.061,21.609,-43.686
C08488=1015.075,-60.263,386.233,-24.060,21.609,-43.691
C08489=1015.075,-60.599,386.258,-24.060,21.610,-43.695
C08490=1015.074,-60.937,386.284,-24.059,21.610,-43.700
C08491=1015.073,-61.275,386.309,-24.059,21.611,-43.706
C08492=1015.072,-61.613,386.335,-24.058,21.611,-43.710
C08493=1015.071,-61.951,386.360,-24.057,21.612,-43.715
C08494=1015.070,-62.290,386.386,-24.057,21.612,-43.720
C08495=1015.069,-62.630,386.411,-24.056,21.614,-43.725
C08496=1015.068,-62.969,386.437,-24.055,21.613,-43.730
C08497=1015.066,-63.309,386.462,-24.055,21.614,-43.735
C08498=1015.065,-63.650,386.487,-24.054,21.615,-43.739
C08499=1015.064,-63.990,386.513,-24.053,21.616,-43.745
C08500=1015.063,-64.331,386.539,-24.053,21.615,-43.750
C08501=1015.061,-64.672,386.565,-24.052,21.617,-43.754
C08502=1015.060,-65.013,386.590,-24.051,21.617,-43.759
C08503=1015.059,-65.356,386.615,-24.051,21.618,-43.765
C08504=1015.058,-65.698,386.641,-24.050,21.617,-43.770
C08505=1015.057,-66.040,386.667,-24.050,21.619,-43.774
C08506=1015.055,-66.383,386.693,-24.049,21.619,-43.780
C08507=1015.054,-66.726,386.718,-24.048,21.620,-43.785
C08508=1015.053,-67.069,386.744,-24.048,21.620,-43.789
C08509=1015.051,-67.412,386.769,-24.047,21.621,-43.795
C08510=1015.050,-67.755,386.795,-24.046,21.621,-43.800
C08511=1015.048,-68.099,386.820,-24.045,21.622,-43.805
C08512=1015.046,-68.443,386.846,-24.045,21.622,-43.809
C08513=1015.045,-68.786,386.872,-24.044,21.623,-43.815
C08514=1015.043,-69.130,386.897,-24.043,21.623,-43.820
C08515=1015.042,-69.474,386.923,-24.043,21.624,-43.824
C08516=1015.041,-69.818,386.949,-24.042,21.624,-43.829
C08517=1015.040,-70.162,386.974,-24.041,21.625,-43.835
C08518=1015.037,-70.506,387.000,-24.041,21.625,-43.840
C08519=1015.036,-70.850,387.026,-24.040,21.626,-43.844
C08520=1015.034,-71.194,387.052,-24.040,21.627,-43.850
C08521=1015.032,-71.538,387.077,-24.039,21.627,-43.855
C08522=1015.031,-71.882,387.103,-24.038,21.628,-43.861
C08523=1015.029,-72.226,387.128,-24.038,21.628,-43.865
C08524=1015.027,-72.570,387.154,-24.037,21.629,-43.870
C08525=1015.025,-72.914,387.179,-24.036,21.629,-43.875
C08526=1015.023,-73.258,387.205,-24.035,21.630,-43.881
C08527=1015.022,-73.602,387.230,-24.035,21.630,-43.885
C08528=1015.020,-73.946,387.256,-24.034,21.631,-43.890
C08529=1015.018,-74.290,387.281,-24.033,21.632,-43.896
C08530=1015.016,-74.633,387.306,-24.033,21.632,-43.901
C08531=1015.014,-74.977,387.332,-24.032,21.633,-43.905
C08532=1015.013,-75.321,387.357,-24.031,21.633,-43.911
C08533=1015.011,-75.664,387.383,-24.031,21.634,-43.916
C08534=1015.009,-76.007,387.408,-24.030,21.634,-43.920
C08535=1015.006,-76.349,387.433,-24.030,21.635,-43.926
C08536=1015.005,-76.692,387.458,-24.029,21.635,-43.931
C08537=1015.003,-77.035,387.484,-24.028,21.636,-43.936
C08538=1015.002,-77.377,387.509,-24.028,21.636,-43.940
C08539=1014.999,-77.719,387.534,-24.027,21.637,-43.946
C08540=1014.997,-78.061,387.559,-24.026,21.637,-43.951
C08541=1014.995,-78.402,387.585,-24.026,21.639,-43.955
C08542=1014.993,-78.744,387.610,-24.025,21.638,-43.960
C08543=1014.991,-79.084,387.635,-24.024,21.639,-43.966
C08544=1014.989,-79.425,387.660,-24.023,21.639,-43.971
C08545=1014.986,-79.765,387.685,-24.023,21.641,-43.975
C08546=1014.984,-80.105,387.710,-24.022,21.641,-43.981
C08547=1014.981,-80.444,387.735,-24.021,21.641,-43.986
C08548=1014.979,-80.783,387.760,-24.021,21.643,-43.990
C08549=1014.977,-81.121,387.785,-24.020,21.643,-43.995
C08550=1014.975,-81.460,387.809,-24.020,21.643,-44.001
C08551=1014.973,-81.798,387.834,-24.019,21.644,-44.005
C08552=1014.971,-82.136,387.859,-24.018,21.645,-44.010
C08553=1014.968,-82.472,387.884,-24.018,21.645,-44.016
C08554=1014.966,-82.809,387.908,-24.017,21.645,-44.021
C08555=1014.963,-83.145,387.933,-24.016,21.646,-44.025
C08556=1014.961,-83.481,387.957,-24.016,21.647,-44.031
C08557=1014.959,-83.816,387.982,-24.015,21.647,-44.036
C08558=1014.956,-84.151,388.006,-24.015,21.648,-44.040
C08559=1014.954,-84.485,388.031,-24.014,21.648,-44.045
C08560=1014.951,-84.835,388.056,-24.013,21.649,-44.051
C08561=1014.948,-85.233,388.086,-24.012,21.650,-44.056
C08562=1014.947,-85.444,388.101,-24.012,21.649,-44.060
C08563=1014.945,-85.658,388.117,-24.012,21.649,-44.062
C08564=1014.942,-86.067,388.147,-24.011,21.650,-44.067
C08565=1014.939,-86.426,388.173,-24.010,21.651,-44.073
C08566=1014.937,-86.756,388.197,-24.009,21.652,-44.078
C08567=1014.935,-87.078,388.221,-24.009,21.652,-44.082
C08568=1014.932,-87.394,388.243,-24.008,21.653,-44.088
C08569=1014.930,-87.707,388.266,-24.007,21.653,-44.093
C08570=1014.927,-88.017,388.289,-24.007,21.654,-44.097
C08571=1014.924,-88.330,388.312,-24.006,21.654,-44.102
C08572=1014.921,-88.649,388.335,-24.006,21.655,-44.106
C08573=1014.918,-89.020,388.362,-24.005,21.656,-44.114
C08574=1014.917,-89.239,388.378,-24.004,21.656,-44.117
C08575=1014.915,-89.473,388.395,-24.004,21.656,-44.119
C08576=1014.913,-89.711,388.412,-24.004,21.656,-44.121
C08577=1014.911,-89.943,388.429,-24.004,21.657,-44.123
C08578=1014.907,-90.348,388.459,-24.003,21.658,-44.130
C08579=1014.905,-90.686,388.483,-24.002,21.658,-44.136
C08580=1014.902,-91.016,388.507,-24.001,21.659,-44.141
C08581=1014.899,-91.345,388.530,-24.001,21.660,-44.145
C08582=1014.896,-91.674,388.555,-24.000,21.660,-44.150
C08583=1014.893,-92.003,388.579,-23.999,21.660,-44.156
C08584=1014.890,-92.331,388.602,-23.999,21.661,-44.160
C08585=1014.888,-92.657,388.626,-23.998,21.662,-44.165
C08586=1014.885,-92.985,388.649,-23.998,21.662,-44.169
C08587=1014.881,-93.311,388.674,-23.997,21.663,-44.175
C08588=1014.878,-93.636,388.697,-23.996,21.663,-44.180
C08589=1014.875,-93.962,388.721,-23.996,21.664,-44.184
C08590=1014.873,-94.286,388.744,-23.995,21.664,-44.189
C08591=1014.870,-94.610,388.767,-23.994,21.665,-44.193
C08592=1014.866,-94.934,388.791,-23.994,21.666,-44.199
C08593=1014.864,-95.258,388.814,-23.993,21.666,-44.204
C08594=1014.860,-95.580,388.838,-23.993,21.666,-44.207
C08595=1014.857,-95.902,388.860,-23.992,21.667,-44.213
C08596=1014.855,-96.225,388.884,-23.991,21.668,-44.217
C08597=1014.851,-96.546,388.907,-23.991,21.668,-44.222
C08598=1014.848,-96.868,388.931,-23.990,21.669,-44.226
C08599=1014.844,-97.189,388.953,-23.989,21.669,-44.231
C08600=1014.842,-97.509,388.976,-23.989,21.670,-44.236
C08601=1014.839,-97.830,388.999,-23.988,21.670,-44.241
C08602=1014.835,-98.152,389.023,-23.987,21.670,-44.246
C08603=1014.831,-98.472,389.046,-23.987,21.672,-44.250
C08604=1014.828,-98.793,389.069,-23.986,21.671,-44.255
C08605=1014.825,-99.114,389.092,-23.986,21.673,-44.260
C08606=1014.821,-99.435,389.115,-23.985,21.673,-44.265
C08607=1014.818,-99.757,389.138,-23.985,21.673,-44.268
C08608=1014.815,-100.079,389.162,-23.984,21.674,-44.274
C08609=1014.812,-100.400,389.185,-23.983,21.675,-44.278
C08610=1014.809,-100.723,389.207,-23.983,21.675,-44.283
C08611=1014.805,-101.045,389.231,-23.982,21.676,-44.287
C08612=1014.801,-101.368,389.254,-23.981,21.676,-44.292
C08613=1014.797,-101.692,389.277,-23.981,21.677,-44.298
C08614=1014.795,-102.016,389.300,-23.980,21.677,-44.302
C08615=1014.791,-102.341,389.324,-23.980,21.678,-44.307
C08616=1014.788,-102.666,389.347,-23.979,21.679,-44.311
C08617=1014.783,-102.992,389.371,-23.978,21.679,-44.316
C08618=1014.780,-103.318,389.394,-23.978,21.680,-44.320
C08619=1014.776,-103.645,389.417,-23.977,21.680,-44.326
C08620=1014.772,-103.971,389.440,-23.976,21.681,-44.331
C08621=1014.769,-104.299,389.464,-23.976,21.681,-44.335
C08622=1014.765,-104.627,389.487,-23.975,21.681,-44.340
C08623=1014.760,-104.954,389.511,-23.975,21.683,-44.344
C08624=1014.757,-105.282,389.535,-23.974,21.683,-44.350
C08625=1014.753,-105.612,389.558,-23.974,21.684,-44.354
C08626=1014.749,-105.940,389.581,-23.973,21.684,-44.359
C08627=1014.746,-106.269,389.605,-23.972,21.685,-44.365
C08628=1014.742,-106.598,389.628,-23.972,21.685,-44.368
C08629=1014.737,-106.928,389.652,-23.971,21.685,-44.374
C08630=1014.734,-107.257,389.675,-23.971,21.687,-44.378
C08631=1014.730,-107.586,389.699,-23.970,21.687,-44.383
C08632=1014.726,-107.915,389.722,-23.969,21.687,-44.388
C08633=1014.721,-108.244,389.746,-23.969,21.688,-44.392
C08634=1014.717,-108.573,389.770,-23.968,21.689,-44.398
C08635=1014.713,-108.902,389.793,-23.967,21.689,-44.402
C08636=1014.709,-109.230,389.816,-23.967,21.689,-44.407
C08637=1014.705,-109.560,389.840,-23.966,21.690,-44.412
C08638=1014.700,-109.889,389.863,-23.965,21.691,-44.416
C08639=1014.696,-110.217,389.887,-23.965,21.691,-44.422
C08640=1014.693,-110.547,389.910,-23.964,21.692,-44.426
C08641=1014.688,-110.876,389.933,-23.963,21.692,-44.431
C08642=1014.684,-111.204,389.957,-23.963,21.693,-44.436
C08643=1014.679,-111.533,389.980,-23.962,21.693,-44.440
C08644=1014.675,-111.862,390.003,-23.962,21.694,-44.446
C08645=1014.670,-112.191,390.027,-23.961,21.695,-44.449
C08646=1014.666,-112.520,390.051,-23.960,21.695,-44.455
C08647=1014.662,-112.849,390.073,-23.960,21.696,-44.459
C08648=1014.658,-113.177,390.097,-23.959,21.696,-44.464
C08649=1014.652,-113.506,390.121,-23.958,21.697,-44.470
C08650=1014.648,-113.835,390.144,-23.958,21.697,-44.473
C08651=1014.644,-114.163,390.168,-23.957,21.698,-44.479
C08652=1014.639,-114.492,390.191,-23.957,21.699,-44.483
C08653=1014.634,-114.821,390.214,-23.956,21.699,-44.488
C08654=1014.630,-115.150,390.237,-23.956,21.700,-44.492
C08655=1014.626,-115.478,390.261,-23.955,21.700,-44.497
C08656=1014.621,-115.807,390.284,-23.954,21.701,-44.503
C08657=1014.616,-116.136,390.307,-23.954,21.701,-44.507
C08658=1014.611,-116.464,390.330,-23.953,21.701,-44.512
C08659=1014.606,-116.792,390.354,-23.953,21.703,-44.516
C08660=1014.602,-117.121,390.377,-23.952,21.703,-44.521
C08661=1014.596,-117.450,390.400,-23.951,21.704,-44.525
C08662=1014.592,-117.778,390.424,-23.951,21.704,-44.531
C08663=1014.587,-118.107,390.447,-23.950,21.705,-44.535
C08664=1014.582,-118.435,390.470,-23.949,21.705,-44.540
C08665=1014.577,-118.764,390.493,-23.949,21.705,-44.545
C08666=1014.572,-119.092,390.517,-23.948,21.707,-44.549
C08667=1014.568,-119.421,390.540,-23.948,21.707,-44.554
C08668=1014.562,-119.750,390.563,-23.947,21.707,-44.558
C08669=1014.558,-120.078,390.587,-23.946,21.708,-44.564
C08670=1014.552,-120.406,390.609,-23.946,21.709,-44.568
C08671=1014.547,-120.735,390.633,-23.945,21.709,-44.573
C08672=1014.542,-121.063,390.656,-23.945,21.710,-44.577
C08673=1014.537,-121.391,390.679,-23.944,21.710,-44.582
C08674=1014.531,-121.720,390.703,-23.944,21.711,-44.586
C08675=1014.527,-122.048,390.726,-23.943,21.711,-44.591
C08676=1014.521,-122.376,390.749,-23.942,21.712,-44.597
C08677=1014.516,-122.705,390.772,-23.942,21.713,-44.601
C08678=1014.511,-123.034,390.795,-23.941,21.713,-44.606
C08679=1014.506,-123.362,390.818,-23.940,21.714,-44.610
C08680=1014.500,-123.690,390.842,-23.940,21.714,-44.615
C08681=1014.495,-124.018,390.865,-23.939,21.715,-44.620
C08682=1014.489,-124.347,390.888,-23.939,21.715,-44.625
C08683=1014.484,-124.675,390.911,-23.938,21.716,-44.628
C08684=1014.478,-125.003,390.935,-23.937,21.717,-44.634
C08685=1014.473,-125.332,390.958,-23.937,21.717,-44.638
C08686=1014.468,-125.660,390.980,-23.936,21.717,-44.643
C08687=1014.462,-125.988,391.003,-23.936,21.719,-44.647
C08688=1014.457,-126.316,391.027,-23.935,21.719,-44.652
C08689=1014.451,-126.645,391.050,-23.935,21.720,-44.657
C08690=1014.445,-126.973,391.073,-23.934,21.720,-44.662
C08691=1014.439,-127.301,391.096,-23.933,21.720,-44.667
C08692=1014.433,-127.629,391.119,-23.933,21.721,-44.671
C08693=1014.428,-127.957,391.143,-23.932,21.721,-44.676
C08694=1014.422,-128.286,391.166,-23.931,21.722,-44.680
C08695=1014.416,-128.614,391.189,-23.931,21.723,-44.686
C08696=1014.410,-128.942,391.212,-23.930,21.723,-44.689
C08697=1014.405,-129.270,391.235,-23.929,21.723,-44.695
C08698=1014.398,-129.598,391.259,-23.929,21.725,-44.699
C08699=1014.393,-129.926,391.281,-23.928,21.724,-44.704
C08700=1014.387,-130.255,391.304,-23.928,21.726,-44.708
C08701=1014.381,-130.583,391.328,-23.927,21.726,-44.713
C08702=1014.375,-130.911,391.350,-23.927,21.726,-44.717
C08703=1014.368,-131.239,391.374,-23.926,21.727,-44.723
C08704=1014.362,-131.568,391.397,-23.926,21.728,-44.726
C08705=1014.356,-131.895,391.420,-23.925,21.728,-44.732
C08706=1014.350,-132.223,391.443,-23.924,21.729,-44.736
C08707=1014.344,-132.552,391.466,-23.924,21.729,-44.741
C08708=1014.337,-132.880,391.490,-23.923,21.730,-44.745
C08709=1014.332,-133.208,391.512,-23.922,21.731,-44.750
C08710=1014.325,-133.536,391.536,-23.922,21.731,-44.754
C08711=1014.318,-133.864,391.558,-23.921,21.731,-44.759
C08712=1014.312,-134.192,391.582,-23.921,21.732,-44.763
C08713=1014.764,-134.160,391.300,-23.921,21.732,-44.763
C08714=1014.770,-133.831,391.277,-23.921,21.731,-44.759
C08715=1014.776,-133.503,391.255,-23.922,21.731,-44.754
C08716=1014.782,-133.176,391.232,-23.922,21.731,-44.750
C08717=1014.788,-132.847,391.209,-23.923,21.730,-44.745
C08718=1014.793,-132.519,391.186,-23.924,21.729,-44.741
C08719=1014.799,-132.191,391.164,-23.924,21.729,-44.736
C08720=1014.805,-131.863,391.140,-23.925,21.728,-44.732
C08721=1014.810,-131.535,391.118,-23.926,21.728,-44.726
C08722=1014.816,-131.207,391.095,-23.926,21.727,-44.723
C08723=1014.822,-130.878,391.072,-23.927,21.726,-44.717
C08724=1014.827,-130.550,391.049,-23.927,21.726,-44.713
C08725=1014.833,-130.222,391.027,-23.928,21.726,-44.708
C08726=1014.838,-129.895,391.003,-23.928,21.724,-44.704
C08727=1014.844,-129.566,390.981,-23.929,21.725,-44.699
C08728=1014.849,-129.238,390.957,-23.929,21.723,-44.695
C08729=1014.854,-128.910,390.935,-23.930,21.723,-44.689
C08730=1014.860,-128.582,390.912,-23.931,21.723,-44.686
C08731=1014.865,-128.254,390.890,-23.931,21.722,-44.680
C08732=1014.871,-127.925,390.867,-23.932,21.721,-44.676
C08733=1014.876,-127.597,390.843,-23.933,21.721,-44.671
C08734=1014.881,-127.269,390.821,-23.933,21.720,-44.667
C08735=1014.887,-126.941,390.798,-23.934,21.720,-44.662
C08736=1014.891,-126.612,390.775,-23.935,21.720,-44.657
C08737=1014.897,-126.284,390.752,-23.935,21.719,-44.652
C08738=1014.902,-125.957,390.729,-23.936,21.719,-44.647
C08739=1014.908,-125.628,390.706,-23.936,21.717,-44.643
C08740=1014.913,-125.300,390.683,-23.937,21.717,-44.638
C08741=1014.918,-124.972,390.660,-23.937,21.717,-44.634
C08742=1014.923,-124.644,390.637,-23.938,21.716,-44.628
C08743=1014.928,-124.315,390.615,-23.939,21.715,-44.625
C08744=1014.932,-123.986,390.592,-23.939,21.715,-44.620
C08745=1014.938,-123.658,390.569,-23.940,21.714,-44.615
C08746=1014.943,-123.330,390.546,-23.940,21.714,-44.610
C08747=1014.948,-123.002,390.523,-23.941,21.713,-44.606
C08748=1014.953,-122.674,390.500,-23.942,21.713,-44.601
C08749=1014.957,-122.345,390.477,-23.942,21.712,-44.597
C08750=1014.962,-122.017,390.454,-23.943,21.711,-44.591
C08751=1014.967,-121.689,390.431,-23.944,21.711,-44.586
C08752=1014.972,-121.360,390.408,-23.944,21.710,-44.582
C08753=1014.977,-121.032,390.385,-23.945,21.710,-44.577
C08754=1014.981,-120.704,390.362,-23.945,21.709,-44.573
C08755=1014.986,-120.374,390.339,-23.946,21.709,-44.568
C08756=1014.991,-120.046,390.316,-23.946,21.708,-44.564
C08757=1014.996,-119.717,390.292,-23.947,21.707,-44.558
C08758=1015.001,-119.389,390.270,-23.948,21.707,-44.554
C08759=1015.006,-119.061,390.247,-23.948,21.707,-44.549
C08760=1015.010,-118.732,390.224,-23.949,21.705,-44.545
C08761=1015.015,-118.404,390.201,-23.949,21.705,-44.540
C08762=1015.019,-118.075,390.177,-23.950,21.705,-44.535
C08763=1015.024,-117.747,390.154,-23.951,21.704,-44.531
C08764=1015.028,-117.418,390.131,-23.951,21.704,-44.525
C08765=1015.033,-117.090,390.108,-23.952,21.703,-44.521
C08766=1015.037,-116.762,390.086,-23.953,21.703,-44.516
C08767=1015.041,-116.434,390.062,-23.953,21.701,-44.512
C08768=1015.046,-116.105,390.040,-23.954,21.701,-44.507
C08769=1015.050,-115.776,390.016,-23.954,21.701,-44.503
C08770=1015.054,-115.448,389.993,-23.955,21.700,-44.497
C08771=1015.059,-115.119,389.970,-23.956,21.700,-44.492
C08772=1015.063,-114.790,389.947,-23.956,21.699,-44.488
C08773=1015.067,-114.462,389.923,-23.957,21.699,-44.483
C08774=1015.072,-114.133,389.901,-23.957,21.698,-44.479
C08775=1015.076,-113.804,389.877,-23.958,21.697,-44.473
C08776=1015.080,-113.476,389.854,-23.958,21.697,-44.470
C08777=1015.084,-113.146,389.831,-23.959,21.696,-44.464
C08778=1015.089,-112.818,389.808,-23.960,21.696,-44.459
C08779=1015.092,-112.489,389.785,-23.960,21.695,-44.455
C08780=1015.097,-112.160,389.762,-23.961,21.695,-44.449
C08781=1015.101,-111.832,389.738,-23.962,21.694,-44.446
C08782=1015.105,-111.502,389.715,-23.962,21.693,-44.440
C08783=1015.109,-111.174,389.692,-23.963,21.693,-44.436
C08784=1015.113,-110.845,389.668,-23.963,21.692,-44.431
C08785=1015.117,-110.516,389.645,-23.964,21.692,-44.426
C08786=1015.121,-110.187,389.622,-23.965,21.691,-44.422
C08787=1015.125,-109.858,389.599,-23.965,21.691,-44.416
C08788=1015.129,-109.529,389.575,-23.966,21.690,-44.412
C08789=1015.132,-109.200,389.552,-23.967,21.689,-44.407
C08790=1015.136,-108.871,389.529,-23.967,21.689,-44.402
C08791=1015.141,-108.542,389.506,-23.968,21.689,-44.398
C08792=1015.145,-108.214,389.482,-23.969,21.688,-44.392
C08793=1015.148,-107.884,389.459,-23.969,21.687,-44.388
C08794=1015.152,-107.555,389.436,-23.970,21.687,-44.383
C08795=1015.156,-107.227,389.412,-23.971,21.687,-44.378
C08796=1015.160,-106.897,389.389,-23.971,21.685,-44.374
C08797=1015.163,-106.568,389.366,-23.972,21.685,-44.368
C08798=1015.167,-106.239,389.342,-23.972,21.685,-44.365
C08799=1015.171,-105.910,389.319,-23.973,21.684,-44.359
C08800=1015.175,-105.581,389.296,-23.974,21.684,-44.354
C08801=1015.179,-105.253,389.272,-23.974,21.683,-44.350
C08802=1015.182,-104.924,389.249,-23.975,21.683,-44.344
C08803=1015.185,-104.596,389.226,-23.975,21.681,-44.340
C08804=1015.188,-104.268,389.202,-23.976,21.681,-44.335
C08805=1015.193,-103.941,389.179,-23.976,21.681,-44.331
C08806=1015.195,-103.614,389.156,-23.977,21.680,-44.326
C08807=1015.199,-103.288,389.133,-23.978,21.680,-44.320
C08808=1015.202,-102.961,389.109,-23.978,21.679,-44.316
C08809=1015.205,-102.636,389.086,-23.979,21.679,-44.311
C08810=1015.209,-102.311,389.063,-23.980,21.678,-44.307
C08811=1015.213,-101.986,389.040,-23.980,21.677,-44.302
C08812=1015.216,-101.662,389.016,-23.981,21.677,-44.298
C08813=1015.220,-101.339,388.993,-23.981,21.676,-44.292
C08814=1015.222,-101.015,388.970,-23.982,21.676,-44.287
C08815=1015.226,-100.692,388.948,-23.983,21.675,-44.283
C08816=1015.229,-100.370,388.924,-23.983,21.675,-44.278
C08817=1015.232,-100.049,388.901,-23.984,21.674,-44.274
C08818=1015.236,-99.727,388.878,-23.985,21.673,-44.268
C08819=1015.239,-99.405,388.855,-23.985,21.673,-44.265
C08820=1015.242,-99.084,388.832,-23.986,21.673,-44.260
C08821=1015.245,-98.763,388.810,-23.986,21.671,-44.255
C08822=1015.248,-98.442,388.786,-23.987,21.672,-44.250
C08823=1015.251,-98.121,388.763,-23.987,21.670,-44.246
C08824=1015.254,-97.801,388.741,-23.988,21.670,-44.241
C08825=1015.257,-97.479,388.718,-23.989,21.670,-44.236
C08826=1015.260,-97.158,388.694,-23.989,21.669,-44.231
C08827=1015.263,-96.837,388.671,-23.990,21.669,-44.226
C08828=1015.266,-96.516,388.648,-23.991,21.668,-44.222
C08829=1015.269,-96.194,388.625,-23.991,21.668,-44.217
C08830=1015.272,-95.873,388.602,-23.992,21.667,-44.213
C08831=1015.275,-95.550,388.579,-23.993,21.666,-44.207
C08832=1015.278,-95.227,388.556,-23.993,21.666,-44.204
C08833=1015.281,-94.904,388.532,-23.994,21.666,-44.199
C08834=1015.284,-94.580,388.509,-23.994,21.665,-44.193
C08835=1015.286,-94.256,388.486,-23.995,21.664,-44.189
C08836=1015.289,-93.931,388.463,-23.996,21.664,-44.184
C08837=1015.292,-93.606,388.439,-23.996,21.663,-44.180
C08838=1015.295,-93.280,388.415,-23.997,21.663,-44.175
C08839=1015.298,-92.955,388.392,-23.998,21.662,-44.169
C08840=1015.300,-92.628,388.368,-23.998,21.662,-44.165
C08841=1015.303,-92.301,388.345,-23.999,21.661,-44.160
C08842=1015.305,-91.972,388.321,-23.999,21.660,-44.156
C08843=1015.309,-91.644,388.298,-24.000,21.660,-44.150
C08844=1015.311,-91.316,388.274,-24.001,21.660,-44.145
C08845=1015.314,-90.987,388.250,-24.001,21.659,-44.141
C08846=1015.316,-90.657,388.226,-24.002,21.658,-44.136
C08847=1015.319,-90.319,388.202,-24.003,21.658,-44.130
C08848=1015.323,-89.912,388.173,-24.004,21.657,-44.123
C08849=1015.324,-89.682,388.155,-24.004,21.656,-44.121
C08850=1015.326,-89.443,388.139,-24.004,21.656,-44.119
C08851=1015.328,-89.210,388.122,-24.004,21.656,-44.117
C08852=1015.330,-88.991,388.105,-24.005,21.656,-44.114
C08853=1015.333,-88.619,388.078,-24.006,21.655,-44.106
C08854=1015.335,-88.301,388.056,-24.006,21.654,-44.102
C08855=1015.337,-87.988,388.033,-24.007,21.654,-44.097
C08856=1015.340,-87.677,388.010,-24.007,21.653,-44.093
C08857=1015.342,-87.365,387.988,-24.008,21.653,-44.088
C08858=1015.344,-87.049,387.965,-24.009,21.652,-44.082
C08859=1015.346,-86.726,387.942,-24.009,21.652,-44.078
C08860=1015.350,-86.397,387.917,-24.010,21.651,-44.073
C08861=1015.352,-86.037,387.891,-24.011,21.650,-44.067
C08862=1015.354,-85.628,387.862,-24.012,21.649,-44.062
C08863=1015.356,-85.415,387.846,-24.012,21.649,-44.060
C08864=1015.358,-85.202,387.830,-24.012,21.650,-44.056
C08865=1015.361,-84.805,387.802,-24.013,21.649,-44.051
C08866=1015.363,-84.456,387.776,-24.014,21.648,-44.045
C08867=1015.366,-84.121,387.752,-24.015,21.648,-44.040
C08868=1015.367,-83.786,387.728,-24.015,21.647,-44.036
C08869=1015.369,-83.451,387.703,-24.016,21.647,-44.031
C08870=1015.372,-83.116,387.678,-24.016,21.646,-44.025
C08871=1015.374,-82.779,387.654,-24.017,21.645,-44.021
C08872=1015.376,-82.443,387.629,-24.018,21.645,-44.016
C08873=1015.379,-82.106,387.605,-24.018,21.645,-44.010
C08874=1015.381,-81.768,387.579,-24.019,21.644,-44.005
C08875=1015.383,-81.431,387.555,-24.020,21.643,-44.001
C08876=1015.385,-81.092,387.531,-24.020,21.643,-43.995
C08877=1015.387,-80.753,387.505,-24.021,21.643,-43.990
C08878=1015.390,-80.415,387.480,-24.021,21.641,-43.986
C08879=1015.391,-80.076,387.457,-24.022,21.641,-43.981
C08880=1015.394,-79.735,387.431,-24.023,21.641,-43.975
C08881=1015.395,-79.395,387.406,-24.023,21.639,-43.971
C08882=1015.397,-79.054,387.381,-24.024,21.639,-43.966
C08883=1015.399,-78.714,387.356,-24.025,21.638,-43.960
C08884=1015.401,-78.373,387.331,-24.026,21.639,-43.955
C08885=1015.404,-78.031,387.306,-24.026,21.637,-43.951
C08886=1015.405,-77.690,387.280,-24.027,21.637,-43.946
C08887=1015.407,-77.348,387.256,-24.028,21.636,-43.940
C08888=1015.409,-77.005,387.230,-24.028,21.636,-43.936
C08889=1015.411,-76.663,387.206,-24.029,21.635,-43.931
C08890=1015.413,-76.320,387.180,-24.030,21.635,-43.926
C08891=1015.415,-75.977,387.155,-24.030,21.634,-43.920
C08892=1015.417,-75.635,387.130,-24.031,21.634,-43.916
C08893=1015.419,-75.291,387.104,-24.031,21.633,-43.911
C08894=1015.421,-74.947,387.079,-24.032,21.633,-43.905
C08895=1015.422,-74.603,387.053,-24.033,21.632,-43.901
C08896=1015.424,-74.260,387.028,-24.033,21.632,-43.896
C08897=1015.425,-73.917,387.003,-24.034,21.631,-43.890
C08898=1015.427,-73.572,386.977,-24.035,21.630,-43.885
C08899=1015.429,-73.229,386.952,-24.035,21.630,-43.881
C08900=1015.430,-72.885,386.926,-24.036,21.629,-43.875
C08901=1015.432,-72.541,386.901,-24.037,21.629,-43.870
C08902=1015.434,-72.197,386.875,-24.038,21.628,-43.865
C08903=1015.436,-71.853,386.850,-24.038,21.628,-43.861
C08904=1015.437,-71.509,386.824,-24.039,21.627,-43.855
C08905=1015.439,-71.165,386.798,-24.040,21.627,-43.850
C08906=1015.440,-70.821,386.774,-24.040,21.626,-43.844
C08907=1015.442,-70.477,386.748,-24.041,21.625,-43.840
C08908=1015.443,-70.133,386.722,-24.041,21.625,-43.835
C08909=1015.445,-69.818,386.699,-24.042,21.625,-43.830
C08910=1015.446,-69.504,386.675,-24.043,21.624,-43.826
C08911=1015.447,-69.101,386.646,-24.043,21.623,-43.820
C08912=1015.449,-68.757,386.620,-24.044,21.623,-43.815
C08913=1015.451,-68.414,386.595,-24.045,21.622,-43.809
C08914=1015.452,-68.070,386.569,-24.045,21.622,-43.805
C08915=1015.453,-67.726,386.543,-24.046,21.621,-43.800
C08916=1015.455,-67.383,386.518,-24.047,21.621,-43.795
C08917=1015.456,-67.039,386.492,-24.048,21.620,-43.789
C08918=1015.457,-66.696,386.467,-24.048,21.620,-43.785
C08919=1015.458,-66.354,386.441,-24.049,21.619,-43.780
C08920=1015.459,-66.011,386.415,-24.050,21.619,-43.774
C08921=1015.461,-65.668,386.390,-24.050,21.617,-43.770
C08922=1015.462,-65.326,386.365,-24.051,21.618,-43.765
C08923=1015.463,-64.985,386.338,-24.051,21.617,-43.759
C08924=1015.464,-64.643,386.313,-24.052,21.617,-43.754
C08925=1015.465,-64.302,386.288,-24.053,21.615,-43.750
C08926=1015.467,-63.961,386.262,-24.053,21.616,-43.745
C08927=1015.468,-63.620,386.236,-24.054,21.615,-43.739
C08928=1015.469,-63.280,386.211,-24.055,21.614,-43.735
C08929=1015.471,-62.940,386.186,-24.055,21.613,-43.730
C08930=1015.471,-62.601,386.160,-24.056,21.614,-43.725
C08931=1015.473,-62.261,386.135,-24.057,21.612,-43.720
C08932=1015.473,-61.922,386.109,-24.057,21.612,-43.715
C08933=1015.474,-61.583,386.084,-24.058,21.611,-43.710
C08934=1015.475,-61.246,386.058,-24.059,21.611,-43.706
C08935=1015.476,-60.908,386.033,-24.059,21.610,-43.700
C08936=1015.477,-60.571,386.008,-24.060,21.610,-43.695
C08937=1015.478,-60.234,385.982,-24.060,21.609,-43.691
C08938=1015.479,-59.898,385.957,-24.061,21.609,-43.686
C08939=1015.480,-59.562,385.931,-24.062,21.608,-43.680
C08940=1015.481,-59.226,385.906,-24.062,21.608,-43.676
C08941=1015.481,-58.891,385.881,-24.063,21.607,-43.671
C08942=1015.483,-58.555,385.855,-24.064,21.607,-43.666
C08943=1015.483,-58.221,385.831,-24.064,21.606,-43.662
C08944=1015.484,-57.887,385.805,-24.065,21.606,-43.656
C08945=1015.484,-57.553,385.780,-24.066,21.605,-43.652
C08946=1015.486,-57.219,385.754,-24.066,21.604,-43.647
C08947=1015.486,-56.886,385.729,-24.067,21.605,-43.642
C08948=1015.487,-56.553,385.704,-24.068,21.603,-43.637
C08949=1015.488,-56.220,385.679,-24.068,21.603,-43.632
C08950=1015.488,-55.888,385.654,-24.069,21.603,-43.627
C08951=1015.489,-55.554,385.628,-24.070,21.602,-43.623
C08952=1015.490,-55.222,385.603,-24.070,21.602,-43.618
C08953=1015.490,-54.889,385.578,-24.071,21.601,-43.613
C08954=1015.491,-54.557,385.553,-24.072,21.601,-43.608
C08955=1015.491,-54.224,385.527,-24.072,21.600,-43.603
C08956=1015.492,-53.892,385.503,-24.073,21.599,-43.599
C08957=1015.492,-53.560,385.477,-24.074,21.600,-43.594
C08958=1015.493,-53.228,385.452,-24.074,21.598,-43.589
C08959=1015.494,-52.896,385.426,-24.075,21.598,-43.584
C08960=1015.494,-52.563,385.402,-24.075,21.597,-43.579
C08961=1015.494,-52.231,385.376,-24.076,21.597,-43.575
C08962=1015.495,-51.899,385.350,-24.077,21.597,-43.570
C08963=1015.495,-51.566,385.326,-24.077,21.596,-43.566
C08964=1015.496,-51.234,385.300,-24.078,21.596,-43.560
C08965=1015.496,-50.901,385.274,-24.079,21.595,-43.555
C08966=1015.497,-50.569,385.249,-24.079,21.594,-43.551
C08967=1015.497,-50.236,385.224,-24.080,21.595,-43.546
C08968=1015.497,-49.904,385.199,-24.080,21.593,-43.542
C08969=1015.498,-49.572,385.173,-24.081,21.593,-43.536
C08970=1015.498,-49.239,385.148,-24.081,21.592,-43.532
C08971=1015.498,-48.907,385.122,-24.082,21.592,-43.527
C08972=1015.498,-48.575,385.097,-24.083,21.592,-43.522
C08973=1015.499,-48.242,385.072,-24.083,21.591,-43.518
C08974=1015.500,-47.909,385.046,-24.084,21.591,-43.512
C08975=1015.500,-47.577,385.020,-24.085,21.589,-43.508
C08976=1015.500,-47.244,384.995,-24.086,21.589,-43.503
C08977=1015.500,-46.912,384.970,-24.086,21.590,-43.498
C08978=1015.500,-46.580,384.944,-24.087,21.588,-43.494
C08979=1015.500,-46.247,384.919,-24.088,21.588,-43.488
C08980=1015.500,-45.915,384.893,-24.088,21.588,-43.485
C08981=1015.500,-45.582,384.867,-24.089,21.587,-43.479
C08982=1015.500,-45.249,384.842,-24.089,21.586,-43.475
C08983=1015.501,-44.917,384.816,-24.090,21.586,-43.470
C08984=1015.501,-44.585,384.790,-24.091,21.586,-43.465
C08985=1015.501,-44.252,384.765,-24.091,21.585,-43.461
C08986=1015.501,-43.919,384.740,-24.092,21.585,-43.455
C08987=1015.500,-43.587,384.713,-24.092,21.584,-43.451
C08988=1015.500,-43.254,384.689,-24.093,21.583,-43.446
C08989=1015.501,-42.922,384.663,-24.094,21.583,-43.442
C08990=1015.500,-42.588,384.637,-24.094,21.583,-43.437
C08991=1015.501,-42.256,384.611,-24.095,21.582,-43.431
C08992=1015.501,-41.924,384.586,-24.096,21.582,-43.427
C08993=1015.500,-41.591,384.560,-24.096,21.582,-43.422
C08994=1015.500,-41.258,384.534,-24.097,21.580,-43.418
C08995=1015.500,-40.926,384.509,-24.098,21.580,-43.413
C08996=1015.500,-40.593,384.483,-24.098,21.580,-43.409
C08997=1015.500,-40.261,384.457,-24.099,21.579,-43.404
C08998=1015.499,-39.928,384.431,-24.100,21.579,-43.398
C08999=1015.499,-39.595,384.406,-24.100,21.578,-43.394
C09000=1015.499,-39.262,384.379,-24.101,21.578,-43.389
C09001=1015.500,-38.930,384.354,-24.101,21.577,-43.385
C09002=1015.499,-38.597,384.328,-24.102,21.577,-43.380
C09003=1015.499,-38.265,384.302,-24.102,21.576,-43.376
C09004=1015.499,-37.932,384.276,-24.103,21.576,-43.371
C09005=1015.498,-37.599,384.251,-24.104,21.575,-43.366
C09006=1015.498,-37.267,384.225,-24.105,21.575,-43.361
C09007=1015.497,-36.934,384.199,-24.105,21.574,-43.357
C09008=1015.497,-36.601,384.173,-24.106,21.574,-43.352
C09009=1015.497,-36.269,384.147,-24.107,21.574,-43.347
C09010=1015.496,-35.936,384.121,-24.107,21.573,-43.343
C09011=1015.496,-35.603,384.096,-24.108,21.573,-43.337
C09012=1015.496,-35.271,384.070,-24.108,21.572,-43.334
C09013=1015.495,-34.939,384.044,-24.109,21.572,-43.328
C09014=1015.494,-34.605,384.018,-24.109,21.571,-43.324
C09015=1015.494,-34.273,383.992,-24.110,21.571,-43.319
C09016=1015.493,-33.940,383.965,-24.111,21.570,-43.315
C09017=1015.493,-33.607,383.940,-24.111,21.570,-43.310
C09018=1015.493,-33.275,383.914,-24.112,21.569,-43.306
C09019=1015.492,-32.943,383.888,-24.113,21.569,-43.301
C09020=1015.492,-32.609,383.862,-24.113,21.568,-43.296
C09021=1015.492,-32.276,383.836,-24.114,21.568,-43.291
C09022=1015.491,-31.944,383.809,-24.114,21.567,-43.287
C09023=1015.490,-31.611,383.784,-24.115,21.567,-43.282
C09024=1015.490,-31.278,383.758,-24.116,21.566,-43.278
C09025=1015.489,-30.946,383.731,-24.116,21.566,-43.273
C09026=1015.488,-30.612,383.706,-24.117,21.565,-43.269
C09027=1015.488,-30.280,383.679,-24.118,21.565,-43.264
C09028=1015.487,-29.947,383.653,-24.118,21.565,-43.260
C09029=1015.486,-29.614,383.627,-24.119,21.564,-43.254
C09030=1015.485,-29.282,383.601,-24.119,21.563,-43.250
C09031=1015.484,-28.950,383.575,-24.120,21.563,-43.245
C09032=1015.483,-28.616,383.549,-24.120,21.562,-43.241
C09033=1015.483,-28.284,383.523,-24.121,21.562,-43.236
C09034=1015.482,-27.951,383.497,-24.122,21.562,-43.232
C09035=1015.481,-27.618,383.470,-24.123,21.562,-43.227
C09036=1015.480,-27.285,383.444,-24.123,21.560,-43.223
C09037=1015.480,-26.953,383.418,-24.124,21.560,-43.217
C09038=1015.479,-26.620,383.392,-24.124,21.560,-43.214
C09039=1015.478,-26.287,383.365,-24.125,21.559,-43.208
C09040=1015.477,-25.954,383.339,-24.126,21.559,-43.204
C09041=1015.477,-25.622,383.313,-24.126,21.559,-43.199
C09042=1015.475,-25.288,383.287,-24.127,21.558,-43.195
C09043=1015.475,-24.956,383.260,-24.128,21.558,-43.190
C09044=1015.473,-24.623,383.234,-24.128,21.557,-43.186
C09045=1015.473,-24.290,383.208,-24.129,21.557,-43.181
C09046=1015.472,-23.957,383.182,-24.129,21.556,-43.177
C09047=1015.470,-23.625,383.155,-24.130,21.556,-43.171
C09048=1015.469,-23.292,383.130,-24.131,21.555,-43.168
C09049=1015.468,-22.959,383.103,-24.131,21.556,-43.162
C09050=1015.468,-22.627,383.076,-24.132,21.554,-43.158
C09051=1015.466,-22.294,383.050,-24.133,21.554,-43.153
C09052=1015.465,-21.961,383.023,-24.133,21.554,-43.149
C09053=1015.464,-21.628,382.997,-24.134,21.553,-43.144
C09054=1015.463,-21.295,382.970,-24.134,21.552,-43.140
C09055=1015.462,-20.962,382.945,-24.135,21.553,-43.135
C09056=1015.460,-20.630,382.918,-24.136,21.552,-43.131
C09057=1015.459,-20.297,382.891,-24.136,21.551,-43.127
C09058=1015.459,-19.965,382.865,-24.137,21.551,-43.122
C09059=1015.458,-19.792,382.852,-24.137,21.550,-43.118
C09060=1015.456,-19.375,382.818,-24.138,21.550,-43.112
C09061=1015.455,-19.128,382.799,-24.139,21.550,-43.109
C09062=1015.454,-18.866,382.778,-24.139,21.550,-43.107
C09063=1015.453,-18.604,382.757,-24.139,21.549,-43.105
C09064=1015.452,-18.357,382.737,-24.139,21.548,-43.103
C09065=1015.451,-18.135,382.719,-24.140,21.549,-43.100
C09066=1015.450,-17.770,382.691,-24.141,21.548,-43.092
C09067=1015.449,-17.437,382.664,-24.141,21.547,-43.088
C09068=1015.447,-17.104,382.638,-24.142,21.547,-43.083
C09069=1015.446,-16.771,382.611,-24.142,21.547,-43.079
C09070=1015.445,-16.437,382.584,-24.143,21.546,-43.074
C09071=1015.443,-16.103,382.557,-24.144,21.546,-43.070
C09072=1015.442,-15.767,382.531,-24.145,21.546,-43.065
C09073=1015.440,-15.431,382.504,-24.145,21.545,-43.061
C09074=1015.439,-15.093,382.476,-24.146,21.544,-43.055
C09075=1015.438,-14.753,382.449,-24.146,21.544,-43.052
C09076=1015.435,-14.411,382.422,-24.147,21.544,-43.046
C09077=1015.434,-14.067,382.395,-24.147,21.543,-43.042
C09078=1015.432,-13.721,382.367,-24.148,21.543,-43.037
C09079=1015.431,-13.372,382.339,-24.149,21.542,-43.033
C09080=1015.430,-13.022,382.311,-24.149,21.542,-43.028
C09081=1015.428,-12.670,382.283,-24.150,21.541,-43.024
C09082=1015.426,-12.317,382.254,-24.151,21.541,-43.019
C09083=1015.425,-11.962,382.226,-24.151,21.540,-43.014
C09084=1015.423,-11.605,382.198,-24.152,21.540,-43.009
C09085=1015.421,-11.248,382.169,-24.152,21.539,-43.006
C09086=1015.419,-10.889,382.140,-24.153,21.539,-43.000
C09087=1015.418,-10.529,382.111,-24.154,21.539,-42.995
C09088=1015.416,-10.221,382.086,-24.154,21.538,-42.991
C09089=1015.414,-9.859,382.057,-24.155,21.537,-42.987
C09090=1015.411,-9.444,382.024,-24.156,21.537,-42.982
C09091=1015.410,-9.082,381.994,-24.156,21.536,-42.976
C09092=1015.408,-8.718,381.966,-24.157,21.536,-42.971
C09093=1015.405,-8.356,381.936,-24.158,21.536,-42.967
C09094=1015.404,-7.992,381.907,-24.158,21.535,-42.961
C09095=1015.402,-7.626,381.877,-24.159,21.535,-42.956
C09096=1015.400,-7.257,381.848,-24.160,21.534,-42.952
C09097=1015.398,-6.886,381.818,-24.160,21.534,-42.947
C09098=1015.396,-6.511,381.787,-24.161,21.533,-42.941
C09099=1015.394,-6.136,381.757,-24.162,21.533,-42.937
C09100=1015.392,-5.761,381.727,-24.163,21.533,-42.932
C09101=1015.389,-5.387,381.697,-24.163,21.532,-42.928
C09102=1015.388,-5.017,381.667,-24.164,21.532,-42.923
C09103=1015.385,-4.650,381.637,-24.164,21.531,-42.919
C09104=1015.383,-4.289,381.608,-24.165,21.530,-42.913
C09105=1015.380,-3.932,381.579,-24.166,21.531,-42.908
C09106=1015.379,-3.577,381.551,-24.166,21.529,-42.904
C09107=1015.377,-3.225,381.522,-24.167,21.529,-42.899
